# B&R Automation Studio project PT_KB_V01 (part 7)

#### TEHNICKI_DODATAK.md
~~~~markdown
# FLOW CHART MASTER — Rad_PG_KB + BRB2_rad

> Detaljni operativni dijagrami za state mašinu Podstanice Grejanja Kotlarnica Banja (PG_KB)
> i BRB2 (bunar) sa vezama preko AsIMA. Svi substepovi, tranzicije, akcije, timeouti.

---

## A. ASCII P&ID skica (referenca za sve dijagrame)

> **VAŽNO — topologija PG_PV05:** proporcionalni ventil `PG_PV05` je **odvojak PRE** `PG_V02` (ne posle). Odvaja se od dolazne BRB2 magistrale i vodi na drenažni kanal. `PG_V05` je zaseban ON/OFF ventil na bypass grani IEBKB1 — nema nikakve veze sa `PG_PV05`.

```
                    ┌── PG_PV05 ──> DRENAŽNI KANAL
                    │      • ispiranje: čeka T na TT_PG_07 >= 60 °C (SP podesiv sa HMI)
                    │      • održavanje pritiska ≥ 5 bar na potisu BRB2 dok su
                    │        ventili tanka zatvoreni (drži bunar u režimu)
                    │      • održavanje 6–7 bar dok su ventili tanka aktivni
                    │        (rasterećenje ka drenaži — štiti izmenjivače i cev)
                    │      • anti-hidraulički udar: P_dolaz > 6.5 bar → auto open
                    │
BRB2 ulaz ──────────┤
(optika ka BRB2_1)  │
                    │                          ┌─ PG_V06 ─ PG_PV01 ─┐
                    └── PG_V02 ────────────────┤                    ├──> Prihvatni tank
                                               └─ PG_V07 ─ PG_PV02 ─┘         │
                                                                              │  ┌ LS_PG_01 (nivo, SP=1.5m)
                                                                              │  ┌ PTNS_PG_01 (P,T,N)
                                                                              │
IEBKB1 ulaz ──> PG_V01 ──────────────> PG_V05 ────────────────────────────────┤
(optika ka IEBKB1)                    (BYPASS ON/OFF —                        │
                                       aktivan samo u IEBKB1 modu)            │
                                                                              │
                                                                       ┌── PG_V03 ── Pu_PG_01 ──┐
                                                                       │                        ├──> ka potrošačima
                                                                       └── PG_V04 ── Pu_PG_02 ──┘  (SP_PritisakPotisa)
```

**Senzori (logička imena u dokumentu → putanja u kodu):**

| Logičko ime | Putanja u kodu | Namena |
|---|---|---|
| `TT_PG_07` | `PG.Sens.Tt._4` (**NOVI — treba dodati u `PG_Sens_Tt_type`**) | Temperatura na drenažnoj cevi iza `PG_PV05` — uslov za završetak ispiranja (SP = 60 °C, podesiv sa HMI) |
| `PG_PT_dolaz` | `PG.Sens.Pt._1` | Pritisak termalne vode na ulazu u podstanicu (pre `PG_V02`) — uslov za anti-udar |
| `PG_PT_potis` | `PG.Sens.Pt._5` | Pritisak potisa iza pumpi `Pu_PG_01/02` (SP = `SetPritisakPotisa`) |
| `PG_PT_BRB2_potis` | `PG.Sens.Pt._6` | Dodatni transmiter -1..9 bar — pritisak dolazne magistrale iza `PG_V02` (mirror preko IMA ka BRB2) |
| `PG_FT_potis` | `PG.Sens.MP._1` | Protok potisa (za `MinProtok/MaxProtok` granice u varijanti 1) |
| `LS_PG_01` | `PG.Sens.LS._1` | Nizak nivo vode u prihvatnom tanku (SP = 1.5 m ciljno) |
| `PTNS_PG_01` | `PG.Sens.Pt._NS1` + `_NS2` | Pritisak na dnu (`_NS1`) i vrhu (`_NS2`) prihvatnog tanka (za proračun nivoa i P u vazdušnom prostoru) |

**Enumerisani selektori (RETAIN, definisani u [Types.typ](Types.typ)):**

| Selektor | Vrednosti |
|---|---|
| `SelektovaniIzvor` (`E_SelektovaniIzvor`) | `_00_nijedan`, `_01_BRB2`, `_02_IEBKB1` |
| `RegulacionaVarijanta` (`E_RegulacionaVarijanta`) | `_00_neaktivan`, `_01_REG_PRITISAK`, `_02_REG_PROTOK`, `_03_REG_TEMPERATURA` |
| `AktivnaPumpaIzlazTanka` (`E_AktivnaPumpaIzlazTanka`) | `_00_nijedna`, `_01_Pu_PG_01`, `_02_Pu_PG_02` |
| `AktivniPropVentilUlazTanka` (`E_AktivniPropVentilUlazTanka`) | `_00_nijedan`, `_01_PG_PV01`, `_02_PG_PV02` |

---

## B. PG_KB state mašina — detaljni stateDiagram

```mermaid
stateDiagram-v2
    direction TB

    [*] --> PG_00_Stand_By: cold boot (State default)

    state PG_00_Stand_By {
        [*] --> ST00_1
        ST00_1: 00.1 Verifikuj mirovanje sistema
        note right of ST00_1
            svi ventili CLOSED
            sve pumpe STOP
            SpremanZaBrb2 := FALSE
            SpremanZaIebkb1 := FALSE
        end note
    }

    PG_00_Stand_By --> PG_01_Priprema_BRB2: SelektovaniIzvor = _01_BRB2\nAND RegulacionaVarijanta <> _00_neaktivan\nAND KomandaStart
    PG_00_Stand_By --> PG_11_Priprema_IEBKB1: SelektovaniIzvor = _02_IEBKB1\nAND RegulacionaVarijanta <> _00_neaktivan\nAND KomandaStart

    %% ═══════════ GRANA BRB2 ═══════════
    state PG_01_Priprema_BRB2 {
        direction TB
        [*] --> ST01_1

        ST01_1: 01.1 Verifikacija interlockova
        note right of ST01_1
            check: PG_V01 = CLOSED
            check: PG_V06 = CLOSED, PG_V07 = CLOSED
            check: PG_V05 = CLOSED
            check: Pu_PG_01 = STOP, Pu_PG_02 = STOP
            check: PG_V03 = CLOSED, PG_V04 = CLOSED
            timeout 5s → Fault F01_INTERLOCK
        end note

        ST01_1 --> ST01_2: interlockovi OK

        ST01_2: 01.2 Otvaranje BRB2 dolaza + start ispiranja
        note right of ST01_2
            PG_V02 → OPEN
            PG_PV05 → 50% (drenaža otvorena)
            IMA: signal BRB2 = "start bunara u ispiranje modu (FR=20Hz)"
            čekaj potvrdu BRB2.PumpaAktivna = TRUE
            timeout 30s → Fault F02_BRB2_NEODZIVA
        end note

        ST01_2 --> ST01_3: BRB2 pumpa startovala

        ST01_3: 01.3 Čekanje temperature ispiranja
        note right of ST01_3
            monitor: TT_PG_07 >= SetPointMinTempIspiranja (60°C, podesivo sa HMI)
            trajanje ispiranja: obično 2-5 min
            timeout 10 min → Fault F03_ISPIRANJE_TIMEOUT
        end note

        ST01_3 --> ST01_4: T_dren dostigla SP

        ST01_4: 01.4 Preusmerenje na tank
        note right of ST01_4
            AKO AktivniPropVentilUlazTanka = _01_PG_PV01:
                PG_V06 → OPEN
                PG_PV01 → aktivan (regulacija nivoa tanka)
            AKO _02_PG_PV02:
                PG_V07 → OPEN
                PG_PV02 → aktivan
            pauza 2s (stabilizacija)
            PG_PV05 → 0% (zatvori drenažu)
            AKO AktivnaPumpaIzlazTanka = _01_Pu_PG_01:
                PG_V03 → OPEN
                Pu_PG_01 → START sa niskim FR (ramp up)
            AKO _02_Pu_PG_02:
                PG_V04 → OPEN
                Pu_PG_02 → START
        end note

        ST01_4 --> ST01_5: ventili otvoreni, pumpa startovala

        ST01_5: 01.5 Signal spremnosti
        note right of ST01_5
            čekaj: nivo tanka > 1.0 m (75% SP)
            čekaj: pritisak potisa >= 90% SP_PritisakPotisa
            čekaj: nema fault-ova
            SpremanZaBrb2 := TRUE
            IMA: šalji spremnost BRB2
        end note
    }

    PG_01_Priprema_BRB2 --> PG_02_Rad_BRB2: 01.5 OK → prelaz na rad
    PG_01_Priprema_BRB2 --> PG_03_Zaustavljanje_BRB2: Fault ILI KomandaStop

    state PG_02_Rad_BRB2 {
        direction TB
        [*] --> ST02_MAIN

        ST02_MAIN: 02.0 Regularni rad
        note right of ST02_MAIN
            aktivni PG_PV01/PV02 → PID(SetPointNivoTanka=1.5m)
            aktivna Pu_PG_01/02 → PID(SetPritisakPotisa)
            monitor MinProtok/MaxProtok override
            IMA: dvosmerni mirror stanja PG↔BRB2
        end note

        ST02_MAIN --> ST02_ANTI: P_dolaz > SetPointMaxPritisakDolaznaCev (6.5 bar)
        ST02_MAIN --> ST02_ROT: uslov rotacije pumpi (radni sati / manuelni zahtev)

        ST02_ANTI: 02.A Anti-hidraulički udar
        note right of ST02_ANTI
            PG_PV05 → auto otvaranje na drenažu (proporcionalno)
            trajanje: dok P_dolaz > 6.4 bar (histerezis 0.1)
            akcija u pozadini, ne menja stanje
        end note
        ST02_ANTI --> ST02_MAIN: P_dolaz < 6.4 bar (histerezis)

        ST02_ROT: 02.R Rotacija Pu_PG_01 ↔ Pu_PG_02
        note right of ST02_ROT
            OVERLAP tranzicija:
              1. start pratite pumpu na 0 Hz
              2. ramp up nova pumpa
              3. ramp down aktivna pumpa
              4. AktivnaPumpaIzlazTanka := novo
              5. zatvori stari PG_V03/V04
        end note
        ST02_ROT --> ST02_MAIN: rotacija završena
    }

    PG_02_Rad_BRB2 --> PG_03_Zaustavljanje_BRB2: KomandaStop\nILI Fault\nILI SelektovaniIzvor promena

    state PG_03_Zaustavljanje_BRB2 {
        direction TB
        [*] --> ST03_1

        ST03_1: 03.1 Redukcija protoka
        note right of ST03_1
            IMA: signal BRB2 = "ramp down bunara"
            PG_PV01/PV02 → ramp down otvor (5s)
            čekaj: protok < 10% MaxProtok
        end note

        ST03_1 --> ST03_2: protok nizak

        ST03_2: 03.2 Zatvaranje tank grane
        note right of ST03_2
            PG_V06 → CLOSED (ili PG_V07)
            PG_PV01 → 0% (ili PG_PV02)
            pauza 1s
        end note

        ST03_2 --> ST03_3: tank grana zatvorena

        ST03_3: 03.3 Zaustavljanje izlazne pumpe
        note right of ST03_3
            Pu_PG_01 → ramp down (ili Pu_PG_02)
            čekaj: pumpa STOP
            PG_V03 → CLOSED (ili PG_V04)
        end note

        ST03_3 --> ST03_4: izlaz zatvoren

        ST03_4: 03.4 Uslovno zatvaranje BRB2 dolaza
        note right of ST03_4
            AKO SelektovaniIzvor menja se u _02_IEBKB1:
                PG_V02 → CLOSED
                IMA: BRB2 = "stop bunara"
            AKO se izvor ne menja:
                PG_V02 ostaje OPEN (za brz restart)
                IMA: BRB2 = "stop bunara"
        end note
    }

    PG_03_Zaustavljanje_BRB2 --> PG_00_Stand_By: 03.4 OK, izvor se ne menja
    PG_03_Zaustavljanje_BRB2 --> PG_11_Priprema_IEBKB1: 03.4 OK, izvor promenjen u _02_IEBKB1

    %% ═══════════ GRANA IEBKB1 ═══════════
    state PG_11_Priprema_IEBKB1 {
        direction TB
        [*] --> ST11_1

        ST11_1: 11.1 Verifikacija interlockova
        note right of ST11_1
            check: PG_V02 = CLOSED
            check: PG_V06 = CLOSED, PG_V07 = CLOSED
            check: PG_PV05 = 0%
            check: PG_V05 = CLOSED
            check: PG_V03 = CLOSED, PG_V04 = CLOSED
            timeout 5s → Fault F11_INTERLOCK
        end note

        ST11_1 --> ST11_2: interlockovi OK

        ST11_2: 11.2 Otvaranje IEBKB1 grane
        note right of ST11_2
            PG_V01 → OPEN
            pauza 1s
            PG_V05 → OPEN (bypass ka tanku)
            IMA: signal IEBKB1 = "start pumpa sa zadatim protokom"
            čekaj potvrdu IEBKB1.PumpaAktivna
            timeout 30s → Fault F12_IEBKB1_NEODZIVA
        end note

        ST11_2 --> ST11_3: IEBKB1 pumpa startovala

        ST11_3: 11.3 Punjenje tanka
        note right of ST11_3
            monitor: nivo tanka raste
            čekaj: nivo >= 1.0 m (75% SP)
            timeout 5 min → Fault F13_PUNJENJE_TIMEOUT
        end note

        ST11_3 --> ST11_4: nivo dostignut

        ST11_4: 11.4 Start izlaza
        note right of ST11_4
            PG_V03 → OPEN (ili PG_V04)
            Pu_PG_01 → START (ili Pu_PG_02)
            čekaj: pritisak potisa >= 90% SP
            SpremanZaIebkb1 := TRUE
        end note
    }

    PG_11_Priprema_IEBKB1 --> PG_12_Rad_IEBKB1: 11.4 OK
    PG_11_Priprema_IEBKB1 --> PG_13_Zaustavljanje_IEBKB1: Fault ILI KomandaStop

    state PG_12_Rad_IEBKB1 {
        direction TB
        [*] --> ST12_MAIN

        ST12_MAIN: 12.0 Regularni rad IEBKB1
        note right of ST12_MAIN
            IEBKB1 pumpa gura zadati protok
            nivo tanka reguliše se protokom IEBKB1 (bez PG_PV01/PV02)
            PG_V05 stalno OPEN
            Pu_PG_01/02 → PID(SetPritisakPotisa)
            IMA: dvosmerni mirror stanja PG↔IEBKB1
        end note

        ST12_MAIN --> ST12_ROT: uslov rotacije izlaznih pumpi
        ST12_ROT: 12.R Rotacija Pu_PG_01 ↔ Pu_PG_02 (isti OVERLAP)
        ST12_ROT --> ST12_MAIN: rotacija završena
    }

    PG_12_Rad_IEBKB1 --> PG_13_Zaustavljanje_IEBKB1: KomandaStop\nILI Fault\nILI SelektovaniIzvor promena

    state PG_13_Zaustavljanje_IEBKB1 {
        direction TB
        [*] --> ST13_1

        ST13_1: 13.1 Redukcija protoka IEBKB1
        note right of ST13_1
            IMA: signal IEBKB1 = "ramp down pumpe"
            čekaj: protok < 10% MaxProtok
        end note

        ST13_1 --> ST13_2: protok nizak

        ST13_2: 13.2 Zatvaranje bypass
        note right of ST13_2
            PG_V05 → CLOSED
            pauza 1s
        end note

        ST13_2 --> ST13_3: bypass zatvoren

        ST13_3: 13.3 Zaustavljanje izlazne pumpe
        note right of ST13_3
            Pu_PG_01/02 → ramp down + STOP
            PG_V03/V04 → CLOSED
        end note

        ST13_3 --> ST13_4: izlaz zatvoren

        ST13_4: 13.4 Uslovno zatvaranje IEBKB1 dolaza
        note right of ST13_4
            AKO SelektovaniIzvor menja se u _01_BRB2:
                PG_V01 → CLOSED
            AKO se izvor ne menja:
                PG_V01 ostaje OPEN (za brz restart)
            IMA: IEBKB1 = "stop pumpa"
        end note
    }

    PG_13_Zaustavljanje_IEBKB1 --> PG_00_Stand_By: 13.4 OK, izvor se ne menja
    PG_13_Zaustavljanje_IEBKB1 --> PG_01_Priprema_BRB2: 13.4 OK, izvor promenjen u _01_BRB2

    %% ═══════════ AUTO-RESTART ═══════════
    note left of PG_00_Stand_By
        AUTO-RESTART posle nestanka struje:
        - State := PG_00_Stand_By (uvek)
        - Ako RETAIN.SelektovaniIzvor <> _00_nijedan
          I RETAIN.RegulacionaVarijanta <> _00_neaktivan
          → automatski KomandaStart → prelaz na 01/11
        - NE zatvara ventile koji su bili otvoreni pre restart-a
          (Priprema faza to prepoznaje kroz interlock check)
    end note
```

---

## C. BRB2_rad state mašina (podsetnik) — proširena Hotel + IEBKB1 grana

```mermaid
stateDiagram-v2
    direction TB

    [*] --> B00_StandBy: cold boot

    B00_StandBy --> B10_Priprema: KomandaStart (od PG_KB preko IMA)\nILI Priprema_Ispiranje

    state B10_Priprema {
        [*] --> B10_1
        B10_1: 10.1 Verifikacija RB2 interlockova
        B10_1 --> B10_2: OK
        B10_2: 10.2 Otvori RB2_V01 (dolaz sa bunara)
        B10_2 --> B10_3: OK
        B10_3: 10.3 Ispiranje (RB2 strana) - dok T_bunar OK
        B10_3 --> B10_4: T OK
        B10_4: 10.4 Grananje prema Ctrl.OdredisteBRB2
    }

    B10_Priprema --> B20_Rad_Hotel: OdredisteBRB2 = _01_Hotel
    B10_Priprema --> B25_Rad_IEBKB1: OdredisteBRB2 = _02_IEBKB1

    state B20_Rad_Hotel {
        [*] --> B20_1
        B20_1: 20.1 Otvori RB2_V02 (ka Hotelu preko PG)
        B20_1 --> B20_2: OK
        B20_2: 20.2 Ramp up pumpe bunara
        B20_2 --> B20_MAIN: OK
        B20_MAIN: 20.M Regularni rad prema RegulacionaVarijanta
        note right of B20_MAIN
            var _01_PRITISAK: FR = f(P_potis)
            var _02_PROTOK:  FR = f(FT_potis)
            var _03_TEMP:    FR = f(T_sekundar)
            IMA: dvosmerni mirror sa PG_KB
        end note
    }

    state B25_Rad_IEBKB1 {
        [*] --> B25_1
        B25_1: 25.1 Otvori RB2_V03 (ka IEBKB1)
        B25_1 --> B25_2: OK
        B25_2: 25.2 Ramp up pumpe bunara
        B25_2 --> B25_MAIN: OK
        B25_MAIN: 25.M Regularni rad za IEBKB1
        note right of B25_MAIN
            uvek varijanta protok
            FR = f(FT_potis)
        end note
    }

    B20_Rad_Hotel --> B30_Zaustavljanje_Hotel: KomandaStop ILI Fault
    B25_Rad_IEBKB1 --> B35_Zaustavljanje_IEBKB1: KomandaStop ILI Fault

    state B30_Zaustavljanje_Hotel {
        [*] --> B30_1
        B30_1: 30.1 Ramp down pumpa bunara
        B30_1 --> B30_2: FR = 0
        B30_2: 30.2 Zatvori RB2_V02
        B30_2 --> B30_3: OK
        B30_3: 30.3 Kondiciono zatvori RB2_V01
    }

    state B35_Zaustavljanje_IEBKB1 {
        [*] --> B35_1
        B35_1: 35.1 Ramp down pumpa
        B35_1 --> B35_2: FR = 0
        B35_2: 35.2 Zatvori RB2_V03
        B35_2 --> B35_3: OK
        B35_3: 35.3 Kondiciono zatvori RB2_V01
    }

    B30_Zaustavljanje_Hotel --> B00_StandBy
    B35_Zaustavljanje_IEBKB1 --> B00_StandBy

    %% Rotacija BRB2 ↔ BRB1_rez radi u pozadini, ne menja glavno stanje
    note left of B20_Rad_Hotel
        Rotacija BRB2 ↔ BRB1_rez:
        OVERLAP tranzicija, prati radne sate
        Menja Ctrl.AktivnaPumpaBunar bez zaustavljanja
    end note
```

---

## D. IMA komunikacija PG↔BRB2 — swimlane sekvenca (Priprema BRB2)

```mermaid
sequenceDiagram
    participant HMI as HMI Operator
    participant PG as PG_KB (PT_KB_V01)
    participant IMA as AsIMA link (optika)
    participant BRB as BRB2_rad (BRB2_1)

    Note over PG,BRB: Auto-boot ili KomandaStart

    HMI->>PG: Set SelektovaniIzvor=_01_BRB2, RegulacionaVarijanta=_02_REG_PROTOK
    HMI->>PG: Set AktivnaPumpaIzlazTanka=_01_Pu_PG_01
    HMI->>PG: Set AktivniPropVentilUlazTanka=_01_PG_PV01
    HMI->>PG: KomandaStart = TRUE

    PG->>PG: PG_00 → PG_01 (Priprema_BRB2)
    PG->>PG: ST01.1 verifikuj interlockove
    PG->>PG: ST01.2 OPEN PG_V02, PG_PV05=50%
    PG->>IMA: TX: Ctrl.SelektovaniIzvor, Ctrl.RegulacionaVarijanta, KomandaStart_BRB2
    IMA->>BRB: RX: Ctrl update od PG_KB

    BRB->>BRB: B00 → B10 (Priprema BRB2)
    BRB->>BRB: OPEN RB2_V01, start pumpa bunara FR=20Hz
    BRB->>IMA: TX: Status.PumpaAktivna=TRUE, Sens.FR_Bunar=20
    IMA->>PG: RX: Status BRB2

    PG->>PG: ST01.3 čekaj TT_PG_07 >= SetPointMinTempIspiranja (SP)
    PG->>IMA: TX: Sens.TT_PG_07 (svaki ciklus)
    IMA->>BRB: RX: (za HMI vizualizaciju na BRB strani)

    Note over PG: TT_PG_07 dostigla SP
    PG->>PG: ST01.4 OPEN PG_V06, PG_PV01 aktivan
    PG->>PG: ST01.4 CLOSE PG_PV05, OPEN PG_V03, START Pu_PG_01
    PG->>PG: ST01.5 SpremanZaBrb2 := TRUE
    PG->>IMA: TX: Status.SpremanZaBrb2=TRUE
    IMA->>BRB: RX: PG spreman

    BRB->>BRB: B10 → B20 (Rad Hotel) - ramp up FR
    BRB->>IMA: TX: Status.SpremanZaPodstanicu=TRUE

    PG->>PG: PG_01 → PG_02 (Rad BRB2)

    Note over PG,BRB: Regularni rad — sve se šalje na obe strane
    loop svaki ciklus
        PG->>IMA: TX: Sens.NivoTanka, PT_potis, FT_potis, TT_PG_07, PT_dolaz, PT_BRB2_potis
        PG->>IMA: TX: Act.Pu_PG_01_FR, PG_PV01_otvor, PG_PV05_otvor
        IMA->>BRB: RX (za HMI)
        BRB->>IMA: TX: Sens.FR_Bunar, PritisakBunar, ProtokBunar, TempBunar
        BRB->>IMA: TX: Act.Pumpa_bunar_snaga
        IMA->>PG: RX (za HMI)
    end
```

---

## E. Fault dijagram + Recovery putanje

```mermaid
stateDiagram-v2
    direction LR

    state "Normal Operation" as NORMAL {
        [*] --> RAD
        RAD: PG_02 / PG_12 aktivno
    }

    NORMAL --> F_INTERLOCK: interlock check FAIL u Priprema fazi
    NORMAL --> F_IZVOR: BRB2/IEBKB1 nije odgovorio 30s (IMA timeout)
    NORMAL --> F_ISPIRANJE: TT_PG_07 nije dostigla SP u 10 min
    NORMAL --> F_NIVO_HIGH: LS_PG_01 > 2.5 m (prepun tank)
    NORMAL --> F_NIVO_LOW: LS_PG_01 < 0.3 m u toku rada
    NORMAL --> F_PRITISAK_HIGH: P_dolaz > 8 bar u toku rada (iznad anti-udara)
    NORMAL --> F_PUMPA: Pu_PG_01/02 alarm (FB_HV_2LS status)
    NORMAL --> F_KOM_IMA: AsIMA link down > 5s

    state "Fault Handling" as FAULT {
        [*] --> F_KLASIFIKUJ
        F_KLASIFIKUJ: Klasifikuj tip fault-a
        F_KLASIFIKUJ --> F_HITNO: F_PRITISAK_HIGH ILI F_NIVO_HIGH
        F_KLASIFIKUJ --> F_KONTROL: F_INTERLOCK ILI F_IZVOR ILI F_KOM_IMA
        F_KLASIFIKUJ --> F_SOFT: F_ISPIRANJE ILI F_NIVO_LOW ILI F_PUMPA

        F_HITNO: HITNO — bezbedno zaustavljanje
        note right of F_HITNO
            SVI ventili CLOSED odmah
            SVE pumpe STOP odmah
            PG_PV05 OPEN (rasterećenje)
            State := PG_00_Stand_By
            FaultLatched := TRUE
            čeka ResetAllowed
        end note

        F_KONTROL: KONTROLISANO zaustavljanje
        note right of F_KONTROL
            prelaz na PG_03 ili PG_13
            uobičajena sekvenca zaustavljanja
            FaultLatched := TRUE
        end note

        F_SOFT: SOFT recovery
        note right of F_SOFT
            pauza u trenutnom substepu
            timeout retry 3x
            posle 3 neuspeha → F_KONTROL
        end note
    }

    F_INTERLOCK --> FAULT
    F_IZVOR --> FAULT
    F_ISPIRANJE --> FAULT
    F_NIVO_HIGH --> FAULT
    F_NIVO_LOW --> FAULT
    F_PRITISAK_HIGH --> FAULT
    F_PUMPA --> FAULT
    F_KOM_IMA --> FAULT

    FAULT --> NORMAL: ResetAllowed + KomandaReset od HMI

    note left of FAULT
        Sve klase pišu u FaultCode/FaultText
        Sve klase šalju IMA notifikaciju
        HMI dobija zvučni alarm
    end note
```

### E.1 Registar fault kodova (`FaultCode : USINT`)

| Kod | Klasa | Okidač | Akcija oporavka |
|-----|-------|--------|-----------------|
| `F01_INTERLOCK` | KONTROL | Interlock check fail u `PG_01` (BRB2 grana) — neki ventil nije u CLOSED, pumpe rade | Zaustavljanje kroz `PG_03` sekvencu; čeka `KomandaReset` |
| `F02_BRB2_NEODZIVA` | KONTROL | BRB2 pumpa nije potvrdila `PumpaAktivna` u 30 s (IMA timeout u `ST01_2`) | Prelaz `PG_03_Zaustavljanje_BRB2`, IMA notifikacija |
| `F03_ISPIRANJE_TIMEOUT` | SOFT | `TT_PG_07` nije dostigla SP (60 °C) u 10 min | Retry 3× (produžava `T_ispiranje`); posle 3. → KONTROL |
| `F11_INTERLOCK` | KONTROL | Interlock check fail u `PG_11` (IEBKB1 grana) | Zaustavljanje kroz `PG_13`; čeka reset |
| `F12_IEBKB1_NEODZIVA` | KONTROL | IEBKB1 pumpa nije potvrdila aktivnost u 30 s | `PG_13_Zaustavljanje_IEBKB1`, IMA notifikacija |
| `F13_PUNJENJE_TIMEOUT` | SOFT | Nivo tanka nije dostigao 1.0 m u 5 min tokom IEBKB1 punjenja | Retry 3×; posle 3. → KONTROL |
| `F20_NIVO_HIGH` | HITNO | `LS_PG_01` mapiran nivo > 2.5 m (prepun tank) | Svi ventili CLOSED, sve pumpe STOP, `PG_PV05` OPEN, State := `PG_00`, `FaultLatched := TRUE` |
| `F21_NIVO_LOW` | SOFT | `LS_PG_01` < 0.3 m u toku aktivnog rada | Pauza substepa, retry 3×; posle 3. → KONTROL |
| `F30_PRITISAK_HIGH` | HITNO | `PG_PT_dolaz` > 8 bar (iznad anti-udar praga 6.5) | HITNO gašenje kao `F20` |
| `F31_ANTI_UDAR_TRAJE` | SOFT | Anti-udar rasterećenje traje > 60 s bez pada P_dolaz-a | Retry 3×; posle 3. → KONTROL |
| `F40_PUMPA_PG` | SOFT | Alarm `Pu_PG_01/02` (FB_HV_2LS status) — pumpa ne prati komandu | Pauza, retry pokretanja; posle 3. → KONTROL sa rotacijom pumpi ako moguće |
| `F50_KOM_IMA` | KONTROL | AsIMA link down > 5 s | `PG_03/PG_13` kontrolisano gašenje; `FaultLatched` dok se link ne uspostavi + operater ne resetuje |
| `F60_KOM_BRB2` | KONTROL | Prijavljen `BRB2.FaultLatched = TRUE` preko IMA | `PG_03_Zaustavljanje_BRB2` |
| `F70_SENZOR_LOST` | HITNO | `ConfigValid = FALSE` na kritičnom `FBAI01_DI01` (Pt._1/._5/._6, MP._1, Tt._4) | HITNO gašenje |

**Reset uslovi:** `KomandaReset` sa HMI + `ResetAllowed = TRUE` (svi FB-ovi imaju `ResetAllowed` izlaz posle BR_Lib update-a).

---

## F. Mapa `.st` fajlova (nomenklatura per substep)

Predlažem sledeću strukturu (spremno za korak 3):

```
PT_KB_V01/Logical/Rad_PG_KB/
├── Cyclic.st                       (CASE dispečer - samo poziva substepove)
├── Init.st                          (default vrednosti SP-ova na cold boot)
├── Exit.st
├── Types.typ                        ✅ ažurirano
├── Variables.var
├── IEC.prg
└── Substeps/
    ├── PG_00_Stand_By.st
    ├── PG_01_1_Interlockovi.st
    ├── PG_01_2_Otvaranje_Ispiranje.st
    ├── PG_01_3_Cekanje_Temperature.st
    ├── PG_01_4_Preusmerenje_Tank.st
    ├── PG_01_5_Signal_Spreman.st
    ├── PG_02_Rad_BRB2.st
    ├── PG_02_A_Anti_Udar.st
    ├── PG_02_R_Rotacija_Pumpi.st
    ├── PG_03_1_Redukcija_Protoka.st
    ├── PG_03_2_Zatvaranje_Tank.st
    ├── PG_03_3_Zaustavljanje_Pumpe.st
    ├── PG_03_4_Uslovno_Zatvaranje_V02.st
    ├── PG_11_1_Interlockovi.st
    ├── PG_11_2_Otvaranje_Bypass.st
    ├── PG_11_3_Punjenje_Tanka.st
    ├── PG_11_4_Start_Izlaza.st
    ├── PG_12_Rad_IEBKB1.st
    ├── PG_13_1_Redukcija_Protoka.st
    ├── PG_13_2_Zatvaranje_Bypass.st
    ├── PG_13_3_Zaustavljanje_Pumpe.st
    ├── PG_13_4_Uslovno_Zatvaranje_V01.st
    ├── FAULT_Klasifikator.st
    ├── FAULT_Hitno.st
    ├── FAULT_Kontrol.st
    └── FAULT_Soft.st
```

Cyclic.st tada postaje kratak dispatcher:

```pascal
CASE State OF
    PG_00_Stand_By:           PG_00_Stand_By_Body();
    PG_01_Priprema_BRB2:
        CASE Substep OF
            1: PG_01_1_Interlockovi();
            2: PG_01_2_Otvaranje_Ispiranje();
            3: PG_01_3_Cekanje_Temperature();
            4: PG_01_4_Preusmerenje_Tank();
            5: PG_01_5_Signal_Spreman();
        END_CASE;
    (* ... itd ... *)
END_CASE;

(* Fault se poziva iznad state mašine kao gate *)
IF FaultLatched THEN
    FAULT_Klasifikator();
END_IF;
```

---

## G. Sledeći koraci (nakon što potvrdiš dijagrame)

1. ~~**Korak 1**: definicija tipova i strukture upravljačkog konteksta.~~ **✅ URAĐENO**
    `E_RegulacionaVarijanta`, `E_SelektovaniIzvor`, `E_AktivnaPumpaIzlazTanka`, `E_AktivniPropVentilUlazTanka`, `typParPG` i `typCtrlPG` su deo globalnog tipa `PG_type`; paralelno `typBRB2Rad` postoji u [BRB2_1/Logical/Project/BRB2_rad/Types.typ](../../../../BRB2_1/Logical/Project/BRB2_rad/Types.typ). `PG : PG_type` i `BRB2Rad : typBRB2Rad` deklarisani su kao `RETAIN`.
2. ~~**Korak 2**: preusmeriti postojeći `Cyclic.st` da koristi `PG.Ctrl.*` umesto pojedinačnih promenljivih.~~ **✅ URAĐENO** (i za `BRB2_rad/Cyclic.sfc`).
3. **Korak 2.5** (na redu): dopuna [Variables.var](Variables.var):
   - `Substep : USINT := 0` (0 = ulazak u state, 1..N = koraci)
   - `KomandaStart : BOOL`, `KomandaStop : BOOL`, `KomandaReset : BOOL` (sa HMI)
   - `FaultLatched : BOOL`
   - `FaultCode : USINT` (šifre iz sekcije E.1)
   - `FaultText : STRING[80]` (za HMI display)
   - Dodati `T_OverlapPumpi : TIME := T#10s` u `typParPG_KB` u [Types.typ](Types.typ)
4. **Korak 2.6** (paralelno): dodati u `PG_Sens_Tt_type` u [Global.typ](../Global.typ) novo polje `_4 : FBAI01_DI01;` sa komentarom „Temperatura na drenaznoj cevi iza PG_PV05 — TT_PG_07", plus fizičko mapiranje kanala u [IO](../IO/).
5. **Korak 3**: kreirati folder `Substeps/` sa praznim skeletonima svakog substep fajla (imena iz sekcije F).
6. **Korak 4**: kreirati komunikacioni tip `PG_00_Comm_Types.typ` — čisto-podatkovni mirror struct (samo `REAL`/`BOOL`/`INT`, bez FB instanci) za AsIMA prenos u oba smera. Poštuje BR_Lib verzijsku razliku između BRB2_1 i PT_KB_V01.
7. **Korak 5**: implementirati logiku redom (najsigurniji prvo — `PG_00_Stand_By`, pa `PG_01_1_Interlockovi`, itd.).
8. **Korak 6**: sinhronizovati enum ekvivalente i mirror strukture u BRB2_1 (za simetriju IMA).

---

## H. Zatvorena pitanja iz validacije dijagrama

| # | Pitanje | Odluka |
|---|---------|--------|
| 1 | Nazivi senzora (`PG_TT_dren`, `PG_PT_dolaz`…) | Prihvaćeno mapiranje iz sekcije A tabele senzora. Kanonska imena u kodu su `PG.Sens.Pt._N` / `Tt._N` / `MP._1` / `LS._N`; logička imena (`TT_PG_07`, `PG_PT_dolaz`, itd.) su za HMI i dokumentaciju. |
| 2 | Fault klase HITNO / KONTROL / SOFT | Prihvaćeno. Detaljan registar u sekciji E.1. |
| 3 | OVERLAP tranzicija pumpi — parametar? | **Da**, `T_OverlapPumpi : TIME := T#10s` dodaje se u `typParPG_KB` (Korak 2.5). Isto važi za rotaciju bunarskih pumpi u `typParBRB2Rad`. |
| 4 | Tip `Substep` varijable — `USINT` ili posebna enum? | `USINT` (0..255). Numeracija prati oznake u sekciji B (npr. `PG_01_1` → `Substep = 1`). Jednostavnije nego enum po fazi, i kompatibilno sa CASE dispečerom u [Cyclic.st](Cyclic.st). |

---

## I. Trenutno stanje implementacije (baseline)

**Legenda:** ✅ postoji u kodu · 🟡 delimično · ⛔ nedostaje

### I.1 PT_KB_V01 / `Rad_PG_KB`

| Artifakt | Fajl | Status |
|---|---|---|
| `E_PG_KB_State` | [Types.typ](Types.typ) | ✅ |
| `E_RegulacionaVarijanta` | [Types.typ](Types.typ) | ✅ |
| `E_SelektovaniIzvor` | [Types.typ](Types.typ) | ✅ |
| `E_AktivnaPumpaIzlazTanka` | [Types.typ](Types.typ) | ✅ |
| `E_AktivniPropVentilUlazTanka` | [Types.typ](Types.typ) | ✅ |
| `typParPG_KB` (Par) | [Types.typ](Types.typ) | ✅ (nedostaje `T_OverlapPumpi`) |
| `typCtrlPG_KB` (Ctrl) | [Types.typ](Types.typ) | ✅ |
| `typPG_KB` | [Types.typ](Types.typ) | ✅ |
| `PG_KB : typPG_KB` (RETAIN) | [Variables.var](Variables.var) | ✅ |
| `State : E_PG_KB_State` | [Variables.var](Variables.var) | ✅ |
| `Substep : USINT` | [Variables.var](Variables.var) | ⛔ Korak 2.5 |
| `KomandaStart/Stop/Reset : BOOL` | [Variables.var](Variables.var) | ⛔ Korak 2.5 |
| `FaultLatched, FaultCode, FaultText` | [Variables.var](Variables.var) | ⛔ Korak 2.5 |
| `Cyclic.st` koristi `PG.Ctrl.*` | [Cyclic.st](Cyclic.st) | ✅ (samo grananje `SelektovaniIzvor`; nema substep dispečera) |
| Substep dispečer (CASE po substep-u) | [Cyclic.st](Cyclic.st) | ⛔ Korak 3 |
| Substep fajlovi u `Substeps/` | — | ⛔ Korak 3 |

### I.2 PT_KB_V01 / globalni tipovi

| Artifakt | Fajl | Status |
|---|---|---|
| `PG_Sens_Pt_type._1.._6, _NS1/2` | [Global.typ](../Global.typ) | ✅ |
| `PG_Sens_Tt_type._1.._3` | [Global.typ](../Global.typ) | ✅ |
| `PG_Sens_Tt_type._4` (TT_PG_07) | [Global.typ](../Global.typ) | ⛔ Korak 2.6 |
| `PG_Sens_MP_type._1` | [Global.typ](../Global.typ) | ✅ |
| `PG_Sens_LS_type._1.._5` | [Global.typ](../Global.typ) | ✅ |

### I.3 BRB2_1 / `BRB2_rad`

| Artifakt | Fajl | Status |
|---|---|---|
| `E_RegulacionaVarijanta` | `BRB2_1/Logical/Project/BRB2_rad/Types.typ` | ✅ |
| `typParBRB2Rad` / `typCtrlBRB2Rad` / `typBRB2Rad` | `BRB2_1/Logical/Project/BRB2_rad/Types.typ` | ✅ |
| `BRB2Rad : typBRB2Rad` (RETAIN) | `BRB2_1/Logical/Project/BRB2_rad/Variables.var` | ✅ |
| `Cyclic.sfc` koristi `BRB2Rad.Ctrl.OdredisteBRB2` | `BRB2_1/Logical/Project/BRB2_rad/Cyclic.sfc` | ✅ |
| `T_OverlapPumpi` (rotacija bunarskih pumpi) | `typParBRB2Rad` | ⛔ Korak 2.5 |
| SFC koraci sa stvarnom logikom | `BRB2_1/Logical/Project/BRB2_rad/Cyclic.sfc` | 🟡 (koraci definisani, sadržaj prazan) |
| BR_Lib verzija (`FB_HV_2LS`, `FB_DI`, `FB_V_ON_OFF_FB`) | `BRB2_1/Logical/Libraries/BR_Lib` | 🟡 stara — treba upgrade pre AsIMA mirror-a (vidi Korak 4) |

### I.4 AsIMA komunikacija PG ↔ BRB2

| Artifakt | Status |
|---|---|
| Fizička optička veza (hardware) | ✅ |
| AsIMA konfiguracija u AS projektu | ⛔ Korak 4 |
| `PG_00_Comm_Types.typ` (mirror struct) | ⛔ Korak 4 |
| Slanje/prijem po ciklusu iz Cyclic-a | ⛔ Korak 4 |

---
~~~~

#### FLOW_CHART_PITANJA.md
```markdown
# Pitanja za flow chart obe strane (BRB2 + PT_KB_V01)

> Upiši odgovore direktno ispod svakog pitanja (na liniji `Odgovor:`).
> Ono što još nisi odlučio ostavi prazno — o tome ćemo posle razgovarati.
> Kad završiš, samo javi "spremno".

---

## FAZA 3: PT_KB_V01 STRANA, GRANA BRB2

### 3.1 `PG_01_Priprema_BRB2`

Šta se sve mora desiti pre nego što Podstanica "objavi" da je spremna za BRB2 (dozvola BRB2 startu)?

**a) Koji ventili se otvaraju/zatvaraju u pripremi?**
(npr. PG_V01 dolazni od BRB2, PG_V02 ka tanku, PG_V03/PG_V04 na izlazu iz tanka — koji od ovih se dira ovde?)

Odgovor: pojsanio u drugom fajlu

**b) Koja pumpa izlaza iz tanka (Pu_PG_01 ili Pu_PG_02) se startuje u pripremi ili tek u fazi Rad_BRB2?**

Odgovor: sve pojasnjeno kada je tank u rau pupa se pali kad nivo predje preko 1.5 metara a gasi kada nivo padne ispod 0.9 metara - ako odrzava nivo ako odzava pritisak ne interesuje je nivo dok ne padne ispod miniumam onda krece da odrzava taj minimalni nivo

**c) Ima li provera pritiska/temperature pre nego što se izađe iz Priprema?**

Odgovor:odgovrio u drugom fajlu

**d) Koji "OK" signal Podstanica šalje BRB2 strani preko IMA (npr. `PG.Status.SpremanZaBrb2 : BOOL`) — i šta znači?**

Odgovor:odgovreno ranije

---

### 3.2 `PG_02_Rad_BRB2`

Šta radi Podstanica dok BRB2 aktivno gura vodu?

**a) Koja pumpa izlaza iz tanka radi (Pu_PG_01 default? auto rotacija? manual?)**

Odgovor:odogovreno vec

**b) Za trenutno aktivnu Varijantu 2 (BRB2 vodi, PG samo prazni tank do nivoa):**
Koji je "nivo" za regulaciju? Nivo tanka (LT_ senzor)? Pritisak potisa PG pumpe? Nešto treće?

Odgovor:odgovoreno

**c) Šta se dešava sa Varijantom 1 (PG vodi, prati pritisak):**
Ako je aktivna, da li PG šalje "traži više/manje" komandu BRB2 strani preko IMA?

Odgovor:odgovoreno - salje samo nivo i status

**d) Da li se PG_V03/PG_V04 preključuju u toku rada (rotacija pumpe za istrošivost)?**

Odgovor: verovatnio resavacemo kasnije

---

### 3.3 `PG_03_Zaustavljanje_BRB2`

Šta radi Podstanica kada operater (ili sistem) povuče izvor (`SelektovaniIzvor = _00_`)?

**a) Da li Podstanica prvo zaustavlja svoju izlaznu pumpu, pa BRB2 pumpu? Ili obratno? Ili paralelno?**

Odgovor:odgovoreno

**b) Ventili koji se zatvaraju u ovoj fazi — redosled?**

Odgovor: odgovreno ranije

**c) Kada je Zaustavljanje "završeno" — koji su uslovi za povratak u Stand_By?**
(svi ventili zatvoreni? pumpe stopped? pritisak spao ispod X bar?)

Odgovor:odgovreno ranije

---

## FAZA 3.5: PRELAZ Pu_PG_01 ↔ Pu_PG_02

**3.5.a Kako se odlučuje koja pumpa je aktivna?**
Označi ono što važi (obriši ostalo, ili kombinuj):
- [ ] manual (operater sa HMI)
- [ ] auto rotacija po vremenu rada
- [ ] auto rotacija po broju startovanja
- [ ] fallback na drugu ako prva ima alarm
- [ ] kombinacija (dopiši kakva)

Odgovor:odgovreno ranije

**3.5.b Prelaz mora imati "overlap" (obe pumpe rade kratko) ili "hard switch" (jedna se ugasi pre nego druga krene)?**

Odgovor:odgovreno ranije

**3.5.c Ventili PG_V03/PG_V04 — da li se ikad obe drže zatvorene (npr. dok pumpe stoje) ili je barem jedan uvek otvoren?**

Odgovor:odgovreno ranije

---

## FAZA 2: BRB2 STRANA, IEBKB1 GRANA (B25 / B35 / B45)

**2.a Da li je logika ista kao Hotel grana (isti ramp, isti pritisci) samo drugi ventili (RB1_V01 vs RB1_V02, RB2_V01 vs RB2_V02)?**

Odgovor:odgovreno ranije

**2.b Ako je različita — šta se razlikuje?**
(npr. drugi `P_Target`, drugi flush režim, drugi `FR_RampUp`)

Odgovor:nista

**2.c Ispiranje (`IspiranjeAktivno` + PG_PV05) — da li se izvodi za obe grane isto ili samo za Hotel?**

Odgovor:odgovreno ranije

---

## FAZA 4: PT_KB_V01 STRANA, GRANA IEBKB1

**4.a Postoji li već legacy kod (u nekom projektu koji nam nije trenutno otvoren) koji rukuje IEBKB1 stranom sa PT_KB_V01 tačke?**

Odgovor:odgovreno ranije

**4.b Ako ne, samo skiciraj u par rečenica šta se treba desiti (u kojoj se meri razlikuje od BRB2 grane).**

Odgovor:odgovreno ranije

---

## FAULT / PREKIDNE PUTANJE

**F.a Ako se javi kritični fault (npr. LT tanka izgubljen, flow meter izgubljen) u toku `Rad_BRB2` — da li:**
- [ ] sistem preskače direktno u `Zaustavljanje_BRB2` sa normalnom sekvencom
- [ ] postoji zaseban Fault step (`PG_99_Fault`) sa agresivnim gašenjem
- [ ] operater mora ručno da povuče izvor pa da krene normalno gašenje

Odgovor:odgovreno ranije

**F.b Ista pitanja za BRB2 stranu (fault tokom `B30_RadBrb2Hotel`):**

Odgovor:odgovreno ranije

---

## BONUS PITANJE ZA MAPIRANJE

**M.a Da li već imaš fizički nacrtan PID/PFD dijagram procesa (PDF/DWG/scan) koji ti mogu pogledati radi validacije naziva ventila i tokova?**
Ako da, gde ga mogu naći?

Odgovor:odgovreno ranije
```

#### FLOW_CHART_POJASNJENJA.md
~~~~markdown
# Pojašnjenja pre finalnih flow chart-ova

> 6 kratkih pitanja koja su izronila iz tvojih odgovora.
> Popuni pored svakog, snimi, i javi „spremno".

---

## P1. PG_V06 / PG_V07 — potvrda semantike

Iz odgovora zaključujem:
- **PG_V06** = ON/OFF ventil PRE proporcionalnog **PG_PV01**
- **PG_V07** = ON/OFF ventil PRE proporcionalnog **PG_PV02**

Da li je to tačno? Ako nije, kako se zovu i za šta služe?

Odgovor: da tacno je

---

## P2. PG_PV05 — dvostruka uloga?

Do sada je `PG_PV05` bio pomenut kao proporcionalni ventil za **ispiranje/drenažu** (na BRB2 strani, `IspiranjeAktivno`).

Ali sada u odgovoru za pripremu BRB2 kažeš: „pušta se bunar dok voda **na drenaži iza PG_PV05** ne dođe do ~60°C".

Da li je to isti PG_PV05, ili postoji poseban drenažni put? Da li se u pripremi otvara `PG_PV05` na drenažu prema kojem procenatu?

Odgovor:da to je isti venti i on radi isto sto i ventili na ulaz u tank odrzava poritisak na potisu iz BRB2 preko 5 bara uvek ... osim kad su aktivni vetili na ulazu u tank tada on odrzava pritisak na 6 ilio 7 bara i cuva iouzmenjivace i celu liniju od velikog pritiska

---

## P3. Signal PG → BRB2 preko IMA

Šta sve konkretno PG šalje BRB2 strani preko IMA (i obratno)?

Trenutno pretpostavljam PG → BRB2:
- `SpremanZaBrb2 : BOOL`
- `NivoTanka : REAL`
- `RegulacionaVarijanta : E_RegulacionaVarijanta`
- `SelektovaniIzvor : E_SelektovaniIzvor` (ogledalo)

BRB2 → PG:
- `Pt_6_Pressure : REAL` (pritisak dolazne cevi, čita se lokalno u BRB2)
- `Pu_Aktivna : BOOL` (BRB2 pumpa aktivna)
- `FR_Actual : REAL` (trenutna frekvencija BRB2 pumpe)
dodaj i protok ka hotelu
mada je meni ovde biola ideja da se salje sve na obe strane takod a mozes da pridjes izuelizaciji i da ividis i jednu i drugu stranu ....
jer ima protokol je mocan a mi imamo optiku nista necemo ugroziti a dacemo lepu komciju u radu na terenu

Fali/suvišno/preimenovati?

Odgovor: dat gore

---

## P4. Aktivna pumpa BRB2

Rekao si: "postoji logika u kodu kako pumpa radi kada je sistem aktivan, pogledaj, jednostavno je i imaš već i parametre unutra — javi šta si našao".

Našao sam ove parametre u `BRB2_1/Logical/Project/BRB2_rad/Types.typ`:

```
FR_Start        : REAL := 20.0;  (* startna frekvenca [Hz] *)
FR_RampUp       : REAL := 0.5;   (* ramp up [Hz/s] *)
FR_RampDown     : REAL := 0.25;  (* ramp down [Hz/s] *)
T_Zaletanje     : TIME := T#10s; (* pre pocetka podizanja *)
P_Target        : REAL := 5.0;   (* ciljni pritisak Pt_RB2_2 [bar] *)
P_TargetStop    : REAL := 5.2;   (* stop pritisak [bar] *)
FR_MinZeroFlow  : REAL := 0.0;   (* TODO eksperimentalno *)
MinProtok       : REAL;          (* Var1 donja granica *)
MaxProtok       : REAL;          (* Var1 gornja granica *)
SetProtok       : REAL := 6.0;   (* Var2 zadati protok [l/s] *)
```

**Ali gore si u odgovoru 3.1.b rekao "samo treba da se pali selektovana pumpa, sad radi logika samo na pumpu koja je povezana"** — ovo se odnosi na **BRB2 pumpu** (jedna pumpa) ili na **PG izlaz pumpu** (Pu_PG_01/Pu_PG_02)?

Odgovor: odnosi se na PG 01/02

---

## P5. Auto-restart posle nestanka struje

Ovo je važno za dizajn. Predlog:

Kada se PLC probudi:
- `State := PG_00_Stand_By` (uvek?)
- Ili: pročitaj RETAIN `SelektovaniIzvor` i idi u odgovarajući step ako je bio aktivan?

Ako je bio aktivan (npr. `SelektovaniIzvor = _01_BRB2` pre nestanka struje), da li:

- [ ] auto-vrati sistem u `PG_02_Rad_BRB2` bez ponovne pripreme (rizik: ventili u nepoznatom stanju)
- [ ] prođi kroz `PG_01_Priprema_BRB2` sa svim proverama pa u `PG_02_Rad_BRB2`
- [ ] uđi u posebno **Recovery** stanje koje polako obnavlja proces sa proverama pritisaka

Odgovor: vracas se us tanje stand By i pokreces sistem sa preselektovanim ocijama
ne zatvaras PG_PV02 jer se nemanja izvor npr ...

---

## P6. PID dijagram — ponovo pošalji

Rekao si da si mi već poslao PID dijagram. Ako je bio u prethodnoj sesiji, nemam ga trenutno pri ruci.

Molim te:
1. Ubaci ga u chat **kao attachment (slika)** — direktno ću ga pročitati i validirati imena ventila
2. ILI ga stavi u fajl u projektu i reci mi putanju

Odgovor / putanja:

---dodao u prilog

## Šta ću uraditi paralelno (bez čekanja)

Dok odgovaraš, ja radim ovo:

1. **Dodajem `E_AktivniPropVentilUlazTanka` u `typCtrlPG_KB`** (analogno `AktivnaPumpaIzlazTanka`).
2. **Dodajem `SetPointNivoTanka : REAL := 1.5` u `typParPG_KB`**.
3. Pravim **`FLOW_CHART_MASTER.md`** sa mermaid dijagramima:
   - Nadgradnja PG_KB state masine (isti tvoj E_PG_KB_State ali sada sa svim substepima)
   - Isto za BRB2_rad (E_BRB2_State — proširenje trenutnog SFC-a u ST logiku)
   - Sekvenca komunikacije PG↔BRB2 preko IMA
   - Fault putanja + Recovery putanja

Kada odgovoriš na P1–P6, dopunjujem sve rupe i dobijamo finalni dokument koji je „ground truth" za dalju implementaciju.
~~~~

#### FLOW_CHART_POJASNJENJA_2.md
~~~~markdown
# Poslednje mikro-nejasnoće pre finalnog dijagrama

> Popuni pored svakog, snimi, javi "spremno" — pa krećem sa flow chartom.

---

## ISPRAVLJENO RAZUMEVANJE (posle korisnikovih korekcija)

- **PG_PV05** = proporcionalni ventil DIREKTNO na drenažnoj grani (nema ON/OFF ventila pre njega). Uloge:
  - početno **ispiranje** cevi (dok voda ne postigne 60°C na drenaži)
  - **zaštita od hidrauličkih udara** / rasterećenje visokog pritiska (prag ~6.5 bar)
- **PG_V05** = ON/OFF ventil na potpuno posebnoj **bypass grani** za IEBKB1 mod (zaobilazi PG_PV01/PV02, pušta direktno u tank). NEMA VEZE sa PG_PV05.

Topologija:
```
                          ┌── PG_PV05 ──> DRENAŽA
BRB2 ulaz ──> PG_V02 ─────┼── PG_V06 ──> PG_PV01 ──> tank
                          └── PG_V07 ──> PG_PV02 ──> tank
                                                       ▲
IEBKB1 ulaz ──> PG_V01 ────────────> PG_V05 ───────────┘  (bypass)
```pg PV05 se odvaja pre dolaka BRB2 do PG_V02 pogledaj PID !!! ipravi to

---

## PZ1. Anti-udar prag za PG_PV05

Rekao si "6.5 bar". Interpretiram kao: kada pritisak u dolaznoj magistrali (posle PG_V02) pređe 6.5 bar, PG_PV05 se automatski otvara na drenažu radi rasterećenja.

Odgovor: 6.5 Bara

---

## PZ2. PG_V05 — ON/OFF ventil (iz IEBKB1 odgovora)

U odgovoru za IEBKB1 granu si rekao: "otvaraš PG_V01 i PG_V05".

Na PID-u vidim `PG_V05` blizu tanka. Da li je to:
- ON/OFF ventil iza PG_PV05 (posle proporcionalnog, pre ulaska u tank drugim putem)?
- ON/OFF ventil na bypass liniji koja u IEBKB1 modu zaobilazi PG_PV01/PV02?
- Nešto treće?

Kada se otvara PG_V05? U kom modu (samo IEBKB1? i BRB2 nekad?)

Odgovor: - ON/OFF ventil na bypass liniji koja u IEBKB1 modu zaobilazi PG_PV01/PV02?

---

## PZ3. Temperatura drenaže (60°C uslov)

Kada prelaziš sa IEBKB1 na BRB2, BRB2 bunar startuje i "izbacuje" hladnu vodu kroz drenažu dok ne postigne 60°C.

Pitanja:
- Gde je senzor temperature? Koje je ime PG_TT_XX?
- Kroz koji put ide drenaža — kroz PG_PV05 pa gde?
- Koji ventil se otvara na drenažu za vreme grejanja? (Da li je to `PG_V22` sa tanka? Ili nešto drugo?)
- Da li BRB2 pumpa radi u konstantnoj frekvenci tokom ove faze (npr. 20-30 Hz) ili prati neki cilj?

Odgovor: treba das e ugradi objasnio ranije gde se ugradjuje - nbegde na drenaznu cev gde moze da meri temperaturu bode u drenaznoj cevi
Kroz PV05 pa and renzani kanal ucrtano u PID-u i ta temperatura trba da bude SP koji se moze menjati
~~~~

### Program Logical/PG_Intf (IEC)

#### Cyclic.st
```iecst
PROGRAM _CYCLIC
	(* ======================================================================== *)
	(* 1) Lokalni PT-BRB2 procesni ugovor                                       *)
	(* ======================================================================== *)
	PGRad_BRB2.RadKaPodstanici := PGRad_BRB2Cmd.RadKaPodstanici;
	PGRad_BRB2.ManualMode := PGRad_BRB2Cmd.ManualMode;
	PGRad_BRB2.ManualSequence := PGRad_BRB2Cmd.ManualSequence;
	PGRad_BRB2.ManualStart := PGRad_BRB2Cmd.ManualStart;
	PGRad_BRB2.ManualStop := PGRad_BRB2Cmd.ManualStop;
	PGRad_BRB2.ManualNextStep := PGRad_BRB2Cmd.ManualNextStep;
	PGRad_BRB2.ManualAbort := PGRad_BRB2Cmd.ManualAbort;
	PGRad_BRB2.ZahtevStarta := PGRad_BRB2Cmd.ZahtevStarta;
	PGRad_BRB2.ZahtevZaustavljanja := PGRad_BRB2Cmd.ZahtevZaustavljanja;
	PGRad_BRB2.VentiliPodstaniceZatvoreni := PGRad_BRB2Cmd.VentiliPodstaniceZatvoreni;
	PGRad_BRB2.PritisakIEBKB1 := PGRad_BRB2Cmd.PritisakIEBKB1;
	PGRad_BRB2.PodstanicaURezimuRada := PGRad_BRB2Cmd.PodstanicaURezimuRada;

	(* ======================================================================== *)
	(* 2) PT izlazni AsIMA snapshot                                             *)
	(* ======================================================================== *)
	PGRad_BRB2_Tx.RadKaPodstanici := PGRad_BRB2Cmd.RadKaPodstanici;
	PGRad_BRB2_Tx.ManualMode := PGRad_BRB2Cmd.ManualMode;
	PGRad_BRB2_Tx.ManualSequence := PGRad_BRB2Cmd.ManualSequence;
	PGRad_BRB2_Tx.ManualStart := PGRad_BRB2Cmd.ManualStart;
	PGRad_BRB2_Tx.ManualStop := PGRad_BRB2Cmd.ManualStop;
	PGRad_BRB2_Tx.ManualNextStep := PGRad_BRB2Cmd.ManualNextStep;
	PGRad_BRB2_Tx.ManualAbort := PGRad_BRB2Cmd.ManualAbort;
	PGRad_BRB2_Tx.ZahtevStarta := PGRad_BRB2Cmd.ZahtevStarta;
	PGRad_BRB2_Tx.ZahtevZaustavljanja := PGRad_BRB2Cmd.ZahtevZaustavljanja;
	PGRad_BRB2_Tx.VentiliPodstaniceZatvoreni := PGRad_BRB2Cmd.VentiliPodstaniceZatvoreni;
	PGRad_BRB2_Tx.PritisakIEBKB1 := PGRad_BRB2Cmd.PritisakIEBKB1;
	PGRad_BRB2_Tx.PodstanicaURezimuRada := PGRad_BRB2Cmd.PodstanicaURezimuRada;

	(* ======================================================================== *)
	(* 3) BRB2 ulazni procesni status                                           *)
	(* ======================================================================== *)
	PGRad_BRB2.PumpaAktivna := PGRad_BRB2_Rx.PumpaAktivna;
	PGRad_BRB2.IspiranjeProtokDostignut := PGRad_BRB2_Rx.IspiranjeProtokDostignut;
	PGRad_BRB2.IspiranjeMinTrajanjeDostignuto := PGRad_BRB2_Rx.IspiranjeMinTrajanjeDostignuto;
	PGRad_BRB2.StopSPDostignut := PGRad_BRB2_Rx.StopSPDostignut;
	PGRad_BRB2.RB2V01Zatvoren := PGRad_BRB2_Rx.RB2V01Zatvoren;
	PGRad_BRB2.RB2V02Zatvoren := PGRad_BRB2_Rx.RB2V02Zatvoren;
END_PROGRAM
```

#### Exit.st
```iecst
PROGRAM _EXIT
END_PROGRAM
```

#### Init.st
```iecst
PROGRAM _INIT
END_PROGRAM
```

### Program Logical/HMI_Svc (IEC)

#### Init.st - Init code
```iecst
PROGRAM _INIT
	(* ======================================================================== *)
	(* 1) Inicijalizacija Podstanica trend prikaza                              *)
	(* ======================================================================== *)
	PGRad_TrendCursor.Position := 0.5;
	PGRad_TrendCursor.ViewSpan := 14400;
	PGRad_TrendCursor.PreviousViewSpan := 14400;
	PGRad_TrendCursor.FollowNow := TRUE;
	PGRad_TrendCursor.CmdBack := FALSE;
	PGRad_TrendCursor.CmdForward := FALSE;
	PGRad_TrendCursor.CmdNow := FALSE;
END_PROGRAM
```

#### Cyclic.st - Cyclic code
```iecst
PROGRAM _CYCLIC
	(* ======================================================================== *)
	(* 1) Rezim i raspolozivi vremenski opseg Podstanica trenda                 *)
	(* ======================================================================== *)
	(* VC pri otvaranju continuous trenda postavlja mod 1; mod 0 drzi zadati prozor. *)
	PGRad_TrendCursor.AxisMode := 0;

	TrendClock.enable := TRUE;
	TrendClock();
	TrendNow_s := DT_TO_UDINT(TrendClock.DT1);
	IF TrendNow_s > 864000 THEN
		TrendEarliest_s := TrendNow_s - 864000;
	ELSE
		TrendEarliest_s := 0;
	END_IF;
	IF (DT_TO_UDINT(PGRad_TrendCursor.RecordingStart) > TrendEarliest_s)
		AND (DT_TO_UDINT(PGRad_TrendCursor.RecordingStart) <= TrendNow_s) THEN
		TrendEarliest_s := DT_TO_UDINT(PGRad_TrendCursor.RecordingStart);
	END_IF;

	(* ======================================================================== *)
	(* 2) Zoom i navigacija vremenskog prozora                                  *)
	(* ======================================================================== *)
	IF PGRad_TrendCursor.ViewSpan < 3600 THEN
		PGRad_TrendCursor.ViewSpan := 3600;
	ELSIF PGRad_TrendCursor.ViewSpan > 172800 THEN
		PGRad_TrendCursor.ViewSpan := 172800;
	END_IF;

	IF (DT_TO_UDINT(PGRad_TrendCursor.ViewStart) = 0)
		AND (TrendNow_s >= DINT_TO_UDINT(PGRad_TrendCursor.ViewSpan)) THEN
		PGRad_TrendCursor.ViewStart := UDINT_TO_DT(
			TrendNow_s - DINT_TO_UDINT(PGRad_TrendCursor.ViewSpan));
		PGRad_TrendCursor.FollowNow := FALSE;
	END_IF;

	IF PGRad_TrendCursor.ViewSpan <> PGRad_TrendCursor.PreviousViewSpan THEN
		IF PGRad_TrendCursor.FollowNow THEN
			PGRad_TrendCursor.ViewStart := UDINT_TO_DT(
				TrendNow_s - DINT_TO_UDINT(PGRad_TrendCursor.ViewSpan));
		ELSE
			PGRad_TrendCursor.ViewStart := UDINT_TO_DT(
				DT_TO_UDINT(PGRad_TrendCursor.ViewStart)
				+ DINT_TO_UDINT(PGRad_TrendCursor.PreviousViewSpan)
				- DINT_TO_UDINT(PGRad_TrendCursor.ViewSpan));
		END_IF;
		PGRad_TrendCursor.PreviousViewSpan := PGRad_TrendCursor.ViewSpan;
		PGRad_TrendCursor.FollowNow := FALSE;
	END_IF;

	IF PGRad_TrendCursor.CmdNow THEN
		IF TrendNow_s >= DINT_TO_UDINT(PGRad_TrendCursor.ViewSpan) THEN
			PGRad_TrendCursor.ViewStart := UDINT_TO_DT(
				TrendNow_s - DINT_TO_UDINT(PGRad_TrendCursor.ViewSpan));
		END_IF;
		PGRad_TrendCursor.FollowNow := FALSE;
	END_IF;

	IF PGRad_TrendCursor.CmdBack THEN
		PGRad_TrendCursor.FollowNow := FALSE;
		IF DT_TO_UDINT(PGRad_TrendCursor.ViewStart) > (TrendEarliest_s + DINT_TO_UDINT(PGRad_TrendCursor.ViewSpan)) THEN
			PGRad_TrendCursor.ViewStart := UDINT_TO_DT(
				DT_TO_UDINT(PGRad_TrendCursor.ViewStart) - DINT_TO_UDINT(PGRad_TrendCursor.ViewSpan));
		ELSE
			PGRad_TrendCursor.ViewStart := UDINT_TO_DT(TrendEarliest_s);
		END_IF;
	END_IF;

	IF PGRad_TrendCursor.CmdForward THEN
		IF (DT_TO_UDINT(PGRad_TrendCursor.ViewStart) + (2 * DINT_TO_UDINT(PGRad_TrendCursor.ViewSpan))) >= TrendNow_s THEN
			PGRad_TrendCursor.ViewStart := UDINT_TO_DT(
				TrendNow_s - DINT_TO_UDINT(PGRad_TrendCursor.ViewSpan));
			PGRad_TrendCursor.FollowNow := FALSE;
		ELSE
			PGRad_TrendCursor.ViewStart := UDINT_TO_DT(
				DT_TO_UDINT(PGRad_TrendCursor.ViewStart) + DINT_TO_UDINT(PGRad_TrendCursor.ViewSpan));
		END_IF;
	END_IF;

	(* ======================================================================== *)
	(* 3) Oznake vremenske ose i apsolutno vreme kursora                        *)
	(* ======================================================================== *)
	PGRad_TrendCursor.AxisTime0 := PGRad_TrendCursor.ViewStart;
	PGRad_TrendCursor.AxisTime1 := UDINT_TO_DT(
		DT_TO_UDINT(PGRad_TrendCursor.ViewStart) + (DINT_TO_UDINT(PGRad_TrendCursor.ViewSpan) / 8));
	PGRad_TrendCursor.AxisTime2 := UDINT_TO_DT(
		DT_TO_UDINT(PGRad_TrendCursor.ViewStart) + ((2 * DINT_TO_UDINT(PGRad_TrendCursor.ViewSpan)) / 8));
	PGRad_TrendCursor.AxisTime3 := UDINT_TO_DT(
		DT_TO_UDINT(PGRad_TrendCursor.ViewStart) + ((3 * DINT_TO_UDINT(PGRad_TrendCursor.ViewSpan)) / 8));
	PGRad_TrendCursor.AxisTime4 := UDINT_TO_DT(
		DT_TO_UDINT(PGRad_TrendCursor.ViewStart) + ((4 * DINT_TO_UDINT(PGRad_TrendCursor.ViewSpan)) / 8));
	PGRad_TrendCursor.AxisTime5 := UDINT_TO_DT(
		DT_TO_UDINT(PGRad_TrendCursor.ViewStart) + ((5 * DINT_TO_UDINT(PGRad_TrendCursor.ViewSpan)) / 8));
	PGRad_TrendCursor.AxisTime6 := UDINT_TO_DT(
		DT_TO_UDINT(PGRad_TrendCursor.ViewStart) + ((6 * DINT_TO_UDINT(PGRad_TrendCursor.ViewSpan)) / 8));
	PGRad_TrendCursor.AxisTime7 := UDINT_TO_DT(
		DT_TO_UDINT(PGRad_TrendCursor.ViewStart) + ((7 * DINT_TO_UDINT(PGRad_TrendCursor.ViewSpan)) / 8));
	PGRad_TrendCursor.AxisTime8 := UDINT_TO_DT(
		DT_TO_UDINT(PGRad_TrendCursor.ViewStart) + DINT_TO_UDINT(PGRad_TrendCursor.ViewSpan));

	(* VC vraca vreme kursora u ms od pocetka referentnog trend zapisa. *)
	PGRad_TrendCursor.DateTime := UDINT_TO_DT(
		DT_TO_UDINT(PGRad_TrendCursor.RecordingStart)
		+ (PGRad_TrendCursor.Time / 1000));

	PGRad_TrendCursor.CmdBack := FALSE;
	PGRad_TrendCursor.CmdForward := FALSE;
	PGRad_TrendCursor.CmdNow := FALSE;
END_PROGRAM
```

### Package Logical/ProcessUnit - Funkcionalne procesne jedinice.

### Program Logical/ProcessUnit/ProcUnit (IEC)

#### Init.st - Init code
```iecst
PROGRAM _INIT
	(* AirRelease parametri se inicijalizuju u vlasnickom Rad_PG_KB sloju. *)
END_PROGRAM
```

#### Cyclic.st - Cyclic code
```iecst
PROGRAM _CYCLIC
	(* ======================================================================== *)
	(* PROCUNIT - ODZRACIVANJE BR1 I BR2                                     *)
	(* AUTO: FB_AirRelease vodi pritisak i LS stepene.                        *)
	(* MANUAL: EnableManual i ManualSP_Percent daju direktnu servisnu komandu. *)
	(* STOP/FAULT: reset, alarm i bezbedno zatvaranje ostaju u vlasnistvu FB-a. *)
	(* STATUS: State, Alarm, Position i Fault statusi se objavljuju HMI-ju.   *)
	(* ======================================================================== *)
	(* ======================================================================== *)
	(* 1) Izbor parametara odzracivanja prema aktivnom izvoru                   *)
	(* ======================================================================== *)
	IF PGRad_Cmd.AirRelease.UseIEBKB1Parameters THEN
		PGRad_AirRelease.PV03.FB.AR_Param := PGRad.Par.AirRelease.IEBKB1.PV03;
		PGRad_AirRelease.PV04.FB.AR_Param := PGRad.Par.AirRelease.IEBKB1.PV04;
	ELSE
		PGRad_AirRelease.PV03.FB.AR_Param := PGRad.Par.AirRelease.BRB2.PV03;
		PGRad_AirRelease.PV04.FB.AR_Param := PGRad.Par.AirRelease.BRB2.PV04;
	END_IF;

	(* ======================================================================== *)
	(* 2) PV03 odzracivanje ulaza u podstanicu                                  *)
	(* ======================================================================== *)
	PGRad_AirRelease.PV03.FB.AR_Input.Enable := PGRad_Cmd.AirRelease.PV03.Enable;
	PGRad_AirRelease.PV03.FB.AR_Input.EnableManual := PGRad_AirRelease.PV03.Ctrl.EnableManual;
	PGRad_AirRelease.PV03.FB.AR_Input.ManualSP_Percent := PGRad_AirRelease.PV03.Ctrl.ManualSP_Percent;
	PGRad_AirRelease.PV03.FB.AR_Input.Pressure_bar := PG.Sens.Pt._1.AI_Output.ScaledValue;
	PGRad_AirRelease.PV03.FB.AR_Input.LS1_Upper := PG.Sens.LS._3.DI_Output.Value;
	PGRad_AirRelease.PV03.FB.AR_Input.LS2_Middle := PG.Sens.LS._2.DI_Output.Value;
	PGRad_AirRelease.PV03.FB.AR_Input.LS3_Lower := FALSE;
	PGRad_AirRelease.PV03.FB.AR_Input.ResetAlarm :=
		PGRad_Cmd.AirRelease.ResetAll
		OR PGRad_AirRelease.PV03.Ctrl.ResetAlarm
		OR (PT_Alarm.ResetPulse.Devices AND PGRad_AirRelease.PV03.FB.AR_Output.ResetAllowed);
	PGRad_AirRelease.PV03.FB();
	PGRad_AirRelease.PV03.Ctrl.ResetAlarm := FALSE;

	(* ======================================================================== *)
	(* 3) PV04 odzracivanje ulaza u prihvatni tank                              *)
	(* ======================================================================== *)
	PGRad_AirRelease.PV04.FB.AR_Input.Enable := PGRad_Cmd.AirRelease.PV04.Enable;
	PGRad_AirRelease.PV04.FB.AR_Input.EnableManual := PGRad_AirRelease.PV04.Ctrl.EnableManual;
	PGRad_AirRelease.PV04.FB.AR_Input.ManualSP_Percent := PGRad_AirRelease.PV04.Ctrl.ManualSP_Percent;
	PGRad_AirRelease.PV04.FB.AR_Input.Pressure_bar := PG.Sens.Pt._4.AI_Output.ScaledValue;
	PGRad_AirRelease.PV04.FB.AR_Input.LS1_Upper := PG.Sens.LS._5.DI_Output.Value;
	PGRad_AirRelease.PV04.FB.AR_Input.LS2_Middle := PG.Sens.LS._4.DI_Output.Value;
	PGRad_AirRelease.PV04.FB.AR_Input.LS3_Lower := FALSE;
	PGRad_AirRelease.PV04.FB.AR_Input.ResetAlarm :=
		PGRad_Cmd.AirRelease.ResetAll
		OR PGRad_AirRelease.PV04.Ctrl.ResetAlarm
		OR (PT_Alarm.ResetPulse.Devices AND PGRad_AirRelease.PV04.FB.AR_Output.ResetAllowed);
	PGRad_AirRelease.PV04.FB();
	PGRad_AirRelease.PV04.Ctrl.ResetAlarm := FALSE;
END_PROGRAM
```

#### Exit.st - Exit code
```iecst
PROGRAM _EXIT
	(* ProcessUnit nema resurse koje treba zatvarati. *)
END_PROGRAM
```

### Package Logical/IMA_comm_PG_BRB2 - AsIMA master veza podstanice sa BRB2.

### Program Logical/IMA_comm_PG_BRB2/BRB2_com (IEC)

#### Init.st - Init code
```iecst
PROGRAM _INIT
	ResetCommunication := FALSE;
	ResetInProgress := FALSE;
	ResetDone := FALSE;
	ResetFault := FALSE;
	(* ======================================================================== *)
	(* 1) Otvaranje AsIMA master sesije prema BRB2                               *)
	(* ======================================================================== *)
	(* Ime DataObject-a identifikuje AsIMA server BRB2 i vraca stationId sesije. *)
	pDatObjName := ADR('BRB2');
	statusInit := IMAinit(pDatObjName, errorInfo, ADR(stationId));
END_PROGRAM
```

#### Cyclic.st - Cyclic code
```iecst
PROGRAM _CYCLIC
	(* ======================================================================== *)
	(* 1) Priprema i prenos PG01 lokalnog snapshot-a                            *)
	(* ======================================================================== *)
	(* PublishPG01 priprema lokalni AsIMA DTO; IMAcomm obavlja dvosmerni prenos. *)
	IF statusInit = IMA_OK THEN
		PublishPG01;
		statusComm := IMAcomm(stationId, connInfoPV, connInfoAUX);
	END_IF

	(* ======================================================================== *)
	(* 2) Automatsko brisanje komunikacione greske                              *)
	(* ======================================================================== *)
	(* ClearError se zadaje samo dok AsIMA prijavljuje gresku ili povezivanje. *)
	IF (connInfoPV.connectionStatus = IMA_ERROR)
		OR (connInfoPV.connectionStatus = IMA_CONNECTING) THEN
		connInfoPV.commandClearError := 1;
	ELSE
		connInfoPV.commandClearError := 0;
	END_IF

	PG01_Remote := PG01_Remote;
END_PROGRAM
```

#### Exit.st - Exit code
```iecst
PROGRAM _EXIT
	(* ======================================================================== *)
	(* 1) Zatvaranje otvorene AsIMA master sesije                                *)
	(* ======================================================================== *)
	(* Sesija se zatvara samo kada je INIT uspesno dodelio vazeci stationId. *)
	IF stationId <> 0 THEN
		statusClose := IMAclose(stationId);
	END_IF
END_PROGRAM
```

#### Variables.var - Local variables
```iecst
VAR
	(* AsIMA DataObject i identifikator sesije. *)
	pDatObjName : UDINT;       (* Adresa naziva AsIMA DataObject konfiguracije. *)
	stationId : UDINT;         (* Identifikator master AsIMA sesije. *)

	(* Povratni statusi AsIMA poziva. *)
	statusInit : UINT;         (* Rezultat jednokratne AsIMA inicijalizacije. *)
	statusComm : UINT;         (* Rezultat ciklicnog AsIMA prenosa. *)
	statusClose : UINT;        (* Rezultat zatvaranja AsIMA sesije. *)

	(* Dijagnostika inicijalizacije i PV prenosa. *)
	errorInfo : imaInfoStruct; (* Dijagnostika neuspele inicijalizacije. *)
	connInfoPV : imaInfoStruct; (* Status i dijagnostika PV prenosa ka BRB2. *)
	connInfoAUX : imaInfoStruct; (* Status pomocnih AsIMA servisa. *)
	ResetCommunication : BOOL; (* HMI zahtev za ponovno otvaranje AsIMA sesije. *)
	ResetInProgress : BOOL; (* Ponovna inicijalizacija AsIMA sesije je u toku. *)
	ResetDone : BOOL; (* Poslednja HMI reinicijalizacija je uspesno zavrsena. *)
	ResetFault : BOOL; (* Poslednja HMI reinicijalizacija nije uspela. *)
END_VAR
```

#### PublishPG01.st
```iecst
ACTION PublishPG01:
	(* ======================================================================== *)
	(* PUBLISH_PG01 - STATUSNI SNAPSHOT PODSTANICE ZA ASIMA/HMI               *)
	(* AUTO/MANUAL: samo objavljuje izabrane komande i statuse; ne komanduje   *)
	(* lokalnim aktuatorima. STOP/FAULT se prenose kao statusi i kodovi.       *)
	(* ======================================================================== *)
	(* ======================================================================== *)
	(* 1) PG01 kontrolni snapshot za AsIMA DTO                                  *)
	(* ======================================================================== *)
	(* Lokalna stanja se pretvaraju u stabilne brojcane vrednosti komunikacionog ugovora. *)
	(* 1.1) Izabrani izvor termalne vode. *)
	CASE PGRad.Ctrl.SelektovaniIzvor OF
		_01_BRB2: PG01_Local.PGCtrl.Izvor := 1;
		_02_IEBKB1: PG01_Local.PGCtrl.Izvor := 2;
	ELSE
		PG01_Local.PGCtrl.Izvor := 0;
	END_CASE

	(* 1.2) Izabrana regulaciona varijanta izlazne pumpe. *)
	CASE PGRad.Ctrl.RegulacionaVarijanta OF
		_01_REG_PRITISAK: PG01_Local.PGCtrl.Regulacija := 1;
		_02_REG_NIVO: PG01_Local.PGCtrl.Regulacija := 2;
	ELSE
		PG01_Local.PGCtrl.Regulacija := 0;
	END_CASE

	(* 1.3) Izabrana izlazna pumpa prihvatnog tanka. *)
	CASE PGRad.Ctrl.AktivnaPumpaIzlazTanka OF
		_01_Pu_PG_01: PG01_Local.PGCtrl.IzlaznaPumpa := 1;
		_02_Pu_PG_02: PG01_Local.PGCtrl.IzlaznaPumpa := 2;
	ELSE
		PG01_Local.PGCtrl.IzlaznaPumpa := 0;
	END_CASE

	(* 1.4) Aktivni proporcionalni ventil na ulazu tanka. *)
	CASE PGRad.Ctrl.AktivniPropVentilUlazTanka OF
		_01_PG_PV01: PG01_Local.PGCtrl.UlazniPV := 1;
		_02_PG_PV02: PG01_Local.PGCtrl.UlazniPV := 2;
	ELSE
		PG01_Local.PGCtrl.UlazniPV := 0;
	END_CASE

	PG01_Local.PGCtrl.AutoRestart := PGRad.Ctrl.AutoRestart;
	PG01_Local.PGCtrl.State := PGRad_Status.State;
	PG01_Local.PGCtrl.Substep := PGRad_Status.Substep;
	PG01_Local.PGCtrl.Fault := PGRad_Status.Fault;
	PG01_Local.PGCtrl.FaultCode := PGRad_Status.FaultCode;

	(* ======================================================================== *)
	(* 2) PG01 lokalni snapshot za AsIMA sinoptiku                              *)
	(* ======================================================================== *)
	(* 2.1) Pu01: komanda, ostvareni rad, frekvencija i fault prve izlazne pumpe. *)
	PG01_Local.PGAct.Pu01.RunCmd := PG.Act.Pu._1.Start;
	PG01_Local.PGAct.Pu01.Running := PG.Act.Pu._1.Status_inRun;
	PG01_Local.PGAct.Pu01.Frequency := PG.Act.Pu._1.Ostvarena_brzina;
	PG01_Local.PGAct.Pu01.Alarm := PG.Act.Pu._1.Alarm_FR OR PG.Act.Pu._1.Alarm_CAN;

	(* 2.2) Pu02: komanda, ostvareni rad, frekvencija i fault druge izlazne pumpe. *)
	PG01_Local.PGAct.Pu02.RunCmd := PG.Act.Pu._2.Start;
	PG01_Local.PGAct.Pu02.Running := PG.Act.Pu._2.Status_inRun;
	PG01_Local.PGAct.Pu02.Frequency := PG.Act.Pu._2.Ostvarena_brzina;
	PG01_Local.PGAct.Pu02.Alarm := PG.Act.Pu._2.Alarm_FR OR PG.Act.Pu._2.Alarm_CAN;

	(* 2.3) PV01 i PV02: komandovana i stvarna pozicija ulaznih ventila tanka. *)
	PG01_Local.PGAct.PV01.Enable := PG.Act.PV._1.PV_Input.Enable;
	PG01_Local.PGAct.PV01.CmdPercent := PG.Act.PV._1.PV_Output.ActiveSP_Percent;
	PG01_Local.PGAct.PV01.PositionPercent := PG.Act.PV._1.PV_Output.PV_Percent;
	PG01_Local.PGAct.PV01.Alarm := PG.Act.PV._1.PV_Output.FaultActive;
	PG01_Local.PGAct.PV02.Enable := PG.Act.PV._2.PV_Input.Enable;
	PG01_Local.PGAct.PV02.CmdPercent := PG.Act.PV._2.PV_Output.ActiveSP_Percent;
	PG01_Local.PGAct.PV02.PositionPercent := PG.Act.PV._2.PV_Output.PV_Percent;
	PG01_Local.PGAct.PV02.Alarm := PG.Act.PV._2.PV_Output.FaultActive;
	(* 2.4) PV03, PV04 i PV05: lokalni status ostalih proporcionalnih ventila. *)
	PG01_Local.PGAct.PV03.Enable := PG.Act.PV._3.PV_Input.Enable;
	PG01_Local.PGAct.PV03.CmdPercent := PG.Act.PV._3.PV_Output.ActiveSP_Percent;
	PG01_Local.PGAct.PV03.PositionPercent := PG.Act.PV._3.PV_Output.PV_Percent;
	PG01_Local.PGAct.PV03.Alarm := PG.Act.PV._3.PV_Output.FaultActive;
	PG01_Local.PGAct.PV04.Enable := PG.Act.PV._4.PV_Input.Enable;
	PG01_Local.PGAct.PV04.CmdPercent := PG.Act.PV._4.PV_Output.ActiveSP_Percent;
	PG01_Local.PGAct.PV04.PositionPercent := PG.Act.PV._4.PV_Output.PV_Percent;
	PG01_Local.PGAct.PV04.Alarm := PG.Act.PV._4.PV_Output.FaultActive;
	PG01_Local.PGAct.PV05.Enable := PG.Act.PV._5.PV_Input.Enable;
	PG01_Local.PGAct.PV05.CmdPercent := PG.Act.PV._5.PV_Output.ActiveSP_Percent;
	PG01_Local.PGAct.PV05.PositionPercent := PG.Act.PV._5.PV_Output.PV_Percent;
	PG01_Local.PGAct.PV05.Alarm := PG.Act.PV._5.PV_Output.FaultActive;

	(* 2.5) AV01 i AV02: dvosmerne komande i granicni prekidaci dovodnih ventila. *)
	PG01_Local.PGAct.AV01.OpenCmd := PG.Act.AV._1.V_Output.CmdOpen;
	PG01_Local.PGAct.AV01.CloseCmd := PG.Act.AV._1.V_Output.CmdClose;
	PG01_Local.PGAct.AV01.Opened := PG.Act.AV._1.Opened;
	PG01_Local.PGAct.AV01.Closed := PG.Act.AV._1.Closed;
	PG01_Local.PGAct.AV01.Alarm := PG.Act.AV._1.V_Output.FaultLatched;
	PG01_Local.PGAct.AV02.OpenCmd := PG.Act.AV._2.V_Output.CmdOpen;
	PG01_Local.PGAct.AV02.CloseCmd := PG.Act.AV._2.V_Output.CmdClose;
	PG01_Local.PGAct.AV02.Opened := PG.Act.AV._2.Opened;
	PG01_Local.PGAct.AV02.Closed := PG.Act.AV._2.Closed;
	PG01_Local.PGAct.AV02.Alarm := PG.Act.AV._2.V_Output.FaultLatched;
	(* 2.6) AV03 do AV07: zahtev otvaranja, polozaj i fault procesnih ventila. *)
	PG01_Local.PGAct.AV03.OpenCmd := PG.Act.AV._3.Open;
	PG01_Local.PGAct.AV03.Opened := PG.Act.AV._3.Opened;
	PG01_Local.PGAct.AV03.Closed := PG.Act.AV._3.Closed;
	PG01_Local.PGAct.AV03.Alarm := PG.Act.AV._3.V_Output.FaultLatched;
	PG01_Local.PGAct.AV04.OpenCmd := PG.Act.AV._4.Open;
	PG01_Local.PGAct.AV04.Opened := PG.Act.AV._4.Opened;
	PG01_Local.PGAct.AV04.Closed := PG.Act.AV._4.Closed;
	PG01_Local.PGAct.AV04.Alarm := PG.Act.AV._4.V_Output.FaultLatched;
	PG01_Local.PGAct.AV05.OpenCmd := PG.Act.AV._5.Open;
	PG01_Local.PGAct.AV05.Opened := PG.Act.AV._5.Opened;
	PG01_Local.PGAct.AV05.Closed := PG.Act.AV._5.Closed;
	PG01_Local.PGAct.AV05.Alarm := PG.Act.AV._5.V_Output.FaultLatched;
	PG01_Local.PGAct.AV06.OpenCmd := PG.Act.AV._6.Open;
	PG01_Local.PGAct.AV06.Opened := PG.Act.AV._6.Opened;
	PG01_Local.PGAct.AV06.Closed := PG.Act.AV._6.Closed;
	PG01_Local.PGAct.AV06.Alarm := PG.Act.AV._6.V_Output.FaultLatched;
	PG01_Local.PGAct.AV07.OpenCmd := PG.Act.AV._7.Open;
	PG01_Local.PGAct.AV07.Opened := PG.Act.AV._7.Opened;
	PG01_Local.PGAct.AV07.Closed := PG.Act.AV._7.Closed;
	PG01_Local.PGAct.AV07.Alarm := PG.Act.AV._7.V_Output.FaultLatched;
	(* 2.7) RV19 i RV21 do RV27: samo fizicki polozaj i alarm rucnih ventila. *)
	PG01_Local.PGAct.RV19.Opened := PG.Act.RV._19.HV_Output.Opened;
	PG01_Local.PGAct.RV19.Closed := PG.Act.RV._19.HV_Output.Closed;
	PG01_Local.PGAct.RV19.Alarm := PG.Act.RV._19.HV_Output.AlarmLatched;
	PG01_Local.PGAct.RV21.Opened := PG.Act.RV._21.HV_Output.Opened;
	PG01_Local.PGAct.RV21.Closed := PG.Act.RV._21.HV_Output.Closed;
	PG01_Local.PGAct.RV21.Alarm := PG.Act.RV._21.HV_Output.AlarmLatched;
	PG01_Local.PGAct.RV22.Opened := PG.Act.RV._22.HV_Output.Opened;
	PG01_Local.PGAct.RV22.Closed := PG.Act.RV._22.HV_Output.Closed;
	PG01_Local.PGAct.RV22.Alarm := PG.Act.RV._22.HV_Output.AlarmLatched;
	PG01_Local.PGAct.RV23.Opened := PG.Act.RV._23.HV_Output.Opened;
	PG01_Local.PGAct.RV23.Closed := PG.Act.RV._23.HV_Output.Closed;
	PG01_Local.PGAct.RV23.Alarm := PG.Act.RV._23.HV_Output.AlarmLatched;
	PG01_Local.PGAct.RV24.Opened := PG.Act.RV._24.HV_Output.Opened;
	PG01_Local.PGAct.RV24.Closed := PG.Act.RV._24.HV_Output.Closed;
	PG01_Local.PGAct.RV24.Alarm := PG.Act.RV._24.HV_Output.AlarmLatched;
	PG01_Local.PGAct.RV25.Opened := PG.Act.RV._25.HV_Output.Opened;
	PG01_Local.PGAct.RV25.Closed := PG.Act.RV._25.HV_Output.Closed;
	PG01_Local.PGAct.RV25.Alarm := PG.Act.RV._25.HV_Output.AlarmLatched;
	PG01_Local.PGAct.RV26.Opened := PG.Act.RV._26.HV_Output.Opened;
	PG01_Local.PGAct.RV26.Closed := PG.Act.RV._26.HV_Output.Closed;
	PG01_Local.PGAct.RV26.Alarm := PG.Act.RV._26.HV_Output.AlarmLatched;
	PG01_Local.PGAct.RV27.Opened := PG.Act.RV._27.HV_Output.Opened;
	PG01_Local.PGAct.RV27.Closed := PG.Act.RV._27.HV_Output.Closed;
	PG01_Local.PGAct.RV27.Alarm := PG.Act.RV._27.HV_Output.AlarmLatched;

	(* 2.8) Pritisci: vrednost, validnost i fault za svaki analogni Pt kanal. *)
	PG01_Local.PGSens.Pt00.Value := PG.Sens.Pt._0_0.AI_Output.ScaledValue;
	PG01_Local.PGSens.Pt00.Valid := PG.Sens.Pt._0_0.AI_Output.Status;
	PG01_Local.PGSens.Pt00.Alarm := PG.Sens.Pt._0_0.AI_Output.FaultLatched;
	PG01_Local.PGSens.Pt01.Value := PG.Sens.Pt._1.AI_Output.ScaledValue;
	PG01_Local.PGSens.Pt01.Valid := PG.Sens.Pt._1.AI_Output.Status;
	PG01_Local.PGSens.Pt01.Alarm := PG.Sens.Pt._1.AI_Output.FaultLatched;
	PG01_Local.PGSens.Pt02.Value := PG.Sens.Pt._2.AI_Output.ScaledValue;
	PG01_Local.PGSens.Pt02.Valid := PG.Sens.Pt._2.AI_Output.Status;
	PG01_Local.PGSens.Pt02.Alarm := PG.Sens.Pt._2.AI_Output.FaultLatched;
	PG01_Local.PGSens.Pt03.Value := PG.Sens.Pt._3.AI_Output.ScaledValue;
	PG01_Local.PGSens.Pt03.Valid := PG.Sens.Pt._3.AI_Output.Status;
	PG01_Local.PGSens.Pt03.Alarm := PG.Sens.Pt._3.AI_Output.FaultLatched;
	PG01_Local.PGSens.Pt04.Value := PG.Sens.Pt._4.AI_Output.ScaledValue;
	PG01_Local.PGSens.Pt04.Valid := PG.Sens.Pt._4.AI_Output.Status;
	PG01_Local.PGSens.Pt04.Alarm := PG.Sens.Pt._4.AI_Output.FaultLatched;
	PG01_Local.PGSens.Pt05.Value := PG.Sens.Pt._5.AI_Output.ScaledValue;
	PG01_Local.PGSens.Pt05.Valid := PG.Sens.Pt._5.AI_Output.Status;
	PG01_Local.PGSens.Pt05.Alarm := PG.Sens.Pt._5.AI_Output.FaultLatched;
	PG01_Local.PGSens.Pt06.Value := PG.Sens.Pt._6.AI_Output.ScaledValue;
	PG01_Local.PGSens.Pt06.Valid := PG.Sens.Pt._6.AI_Output.Status;
	PG01_Local.PGSens.Pt06.Alarm := PG.Sens.Pt._6.AI_Output.FaultLatched;
	PG01_Local.PGSens.PtNS1.Value := PG.Sens.Pt._NS1.AI_Output.ScaledValue;
	PG01_Local.PGSens.PtNS1.Valid := PG.Sens.Pt._NS1.AI_Output.Status;
	PG01_Local.PGSens.PtNS1.Alarm := PG.Sens.Pt._NS1.AI_Output.FaultLatched;
	PG01_Local.PGSens.PtNS2.Value := PG.Sens.Pt._NS2.AI_Output.ScaledValue;
	PG01_Local.PGSens.PtNS2.Valid := PG.Sens.Pt._NS2.AI_Output.Status;
	PG01_Local.PGSens.PtNS2.Alarm := PG.Sens.Pt._NS2.AI_Output.FaultLatched;
	(* 2.9) Temperature: vrednost, validnost i fault za svaki analogni Tt kanal. *)
	PG01_Local.PGSens.Tt01.Value := PG.Sens.Tt._1.AI_Output.ScaledValue;
	PG01_Local.PGSens.Tt01.Valid := PG.Sens.Tt._1.AI_Output.Status;
	PG01_Local.PGSens.Tt01.Alarm := PG.Sens.Tt._1.AI_Output.FaultLatched;
	PG01_Local.PGSens.Tt02.Value := PG.Sens.Tt._2.AI_Output.ScaledValue;
	PG01_Local.PGSens.Tt02.Valid := PG.Sens.Tt._2.AI_Output.Status;
	PG01_Local.PGSens.Tt02.Alarm := PG.Sens.Tt._2.AI_Output.FaultLatched;
	PG01_Local.PGSens.Tt03.Value := PG.Sens.Tt._3.AI_Output.ScaledValue;
	PG01_Local.PGSens.Tt03.Valid := PG.Sens.Tt._3.AI_Output.Status;
	PG01_Local.PGSens.Tt03.Alarm := PG.Sens.Tt._3.AI_Output.FaultLatched;
	PG01_Local.PGSens.Tt04.Value := PG.Sens.Tt._4.AI_Output.ScaledValue;
	PG01_Local.PGSens.Tt04.Valid := PG.Sens.Tt._4.AI_Output.Status;
	PG01_Local.PGSens.Tt04.Alarm := PG.Sens.Tt._4.AI_Output.FaultLatched;
	PG01_Local.PGSens.Tt05.Value := PG.Sens.Tt._5.AI_Output.ScaledValue;
	PG01_Local.PGSens.Tt05.Valid := PG.Sens.Tt._5.AI_Output.Status;
	PG01_Local.PGSens.Tt05.Alarm := PG.Sens.Tt._5.AI_Output.FaultLatched;
	PG01_Local.PGSens.Tt06.Value := PG.Sens.Tt._6.AI_Output.ScaledValue;
	PG01_Local.PGSens.Tt06.Valid := PG.Sens.Tt._6.AI_Output.Status;
	PG01_Local.PGSens.Tt06.Alarm := PG.Sens.Tt._6.AI_Output.FaultLatched;
	PG01_Local.PGSens.Tt07.Value := PG.Sens.Tt._7.AI_Output.ScaledValue;
	PG01_Local.PGSens.Tt07.Valid := PG.Sens.Tt._7.AI_Output.Status;
	PG01_Local.PGSens.Tt07.Alarm := PG.Sens.Tt._7.AI_Output.FaultLatched;
	PG01_Local.PGSens.Tt08.Value := PG.Sens.Tt._8.AI_Output.ScaledValue;
	PG01_Local.PGSens.Tt08.Valid := PG.Sens.Tt._8.AI_Output.Status;
	PG01_Local.PGSens.Tt08.Alarm := PG.Sens.Tt._8.AI_Output.FaultLatched;
	PG01_Local.PGSens.Tt09.Value := PG.Sens.Tt._9.AI_Output.ScaledValue;
	PG01_Local.PGSens.Tt09.Valid := PG.Sens.Tt._9.AI_Output.Status;
	PG01_Local.PGSens.Tt09.Alarm := PG.Sens.Tt._9.AI_Output.FaultLatched;
	PG01_Local.PGSens.Tt10.Value := PG.Sens.Tt._10.AI_Output.ScaledValue;
	PG01_Local.PGSens.Tt10.Valid := PG.Sens.Tt._10.AI_Output.Status;
	PG01_Local.PGSens.Tt10.Alarm := PG.Sens.Tt._10.AI_Output.FaultLatched;
	PG01_Local.PGSens.Tt11.Value := PG.Sens.Tt._11.AI_Output.ScaledValue;
	PG01_Local.PGSens.Tt11.Valid := PG.Sens.Tt._11.AI_Output.Status;
	PG01_Local.PGSens.Tt11.Alarm := PG.Sens.Tt._11.AI_Output.FaultLatched;
	(* 2.10) MP01: vrednost, validnost i fault merenja nivoa/pritiska. *)
	PG01_Local.PGSens.MP01.Value := PG.Sens.MP._1.AI_Output.ScaledValue;
	PG01_Local.PGSens.MP01.Valid := PG.Sens.MP._1.AI_Output.Status;
	PG01_Local.PGSens.MP01.Alarm := PG.Sens.MP._1.AI_Output.FaultLatched;

	(* 2.11) Digitalni nivo prekidaci i prestrujni ventili: vrednost i alarm. *)
	PG01_Local.PGSens.LS01.Value := PG.Sens.LS._1.DI_Output.Value;
	PG01_Local.PGSens.LS01.Alarm := PG.Sens.LS._1.DI_Output.Alarm;
	PG01_Local.PGSens.LS02.Value := PG.Sens.LS._2.DI_Output.Value;
	PG01_Local.PGSens.LS02.Alarm := PG.Sens.LS._2.DI_Output.Alarm;
	PG01_Local.PGSens.LS03.Value := PG.Sens.LS._3.DI_Output.Value;
	PG01_Local.PGSens.LS03.Alarm := PG.Sens.LS._3.DI_Output.Alarm;
	PG01_Local.PGSens.LS04.Value := PG.Sens.LS._4.DI_Output.Value;
	PG01_Local.PGSens.LS04.Alarm := PG.Sens.LS._4.DI_Output.Alarm;
	PG01_Local.PGSens.LS05.Value := PG.Sens.LS._5.DI_Output.Value;
	PG01_Local.PGSens.LS05.Alarm := PG.Sens.LS._5.DI_Output.Alarm;
	PG01_Local.PGSens.OWF01.Value := PG.Sens.OWF._1.DI_Output.Value;
	PG01_Local.PGSens.OWF01.Alarm := PG.Sens.OWF._1.DI_Output.Alarm;
	PG01_Local.PGSens.OWF02.Value := PG.Sens.OWF._2.DI_Output.Value;
	PG01_Local.PGSens.OWF02.Alarm := PG.Sens.OWF._2.DI_Output.Alarm;
END_ACTION
```

### Data object Logical/IMA_comm_PG_BRB2/BRB2 (Simple)

#### BRB2.dat
```
; AsIMA master configuration: PT_KB_V01 -> BRB2_1
"[ROUTING_PATH]"
"/SECTION=INTERFACE"
"/CN=IF2.19"
"[PV_LIST_1]"
"/SECTION=PV"
"/SV=READ /SERVPV=PGRad_BRB2_Tx /CLNTPV=PGRad_BRB2_Rx"
"/SV=WRITE /SERVPV=PGRad_BRB2_Rx /CLNTPV=PGRad_BRB2_Tx"
"/SV=READ /SERVPV=PG01_Remote /CLNTPV=PG01_Remote"
"/SV=WRITE /SERVPV=PG01_Local /CLNTPV=PG01_Local"
```

### Alarm.typ - not listed in the package file held
```iecst
TYPE
	typAlarmState : STRUCT (* Standardno stanje jednog projektnog alarma. *)
		Active : BOOL; (* TRUE dok je fizicki ili programski uzrok trenutno prisutan. *)
		Latched : BOOL; (* TRUE od prve pojave alarma do dozvoljenog reseta. *)
		Acknowledged : BOOL; (* TRUE nakon operatorske potvrde memorisanog alarma. *)
		ResetAllowed : BOOL; (* TRUE kada aktivni uzrok vise nije prisutan. *)
		Blocking : BOOL; (* TRUE kada alarm blokira novi start ili zahteva kontrolisani stop. *)
		Code : UINT; (* Stabilan projektni alarmni kod. *)
		SourceCode : USINT; (* Lokalni FaultCode izvornog FB-a, kada postoji. *)
		Severity : USINT; (* Prioritet: 1=INFO, 2=WARNING, 3=ALARM, 4=TRIP. *)
	END_STRUCT;

	typAlarmCommand : STRUCT (* Jednociklusne komande projektnog alarmnog sistema. *)
		AcknowledgeAll : BOOL; (* Potvrda svih trenutno memorisanih alarma bez reseta opreme. *)
		ResetAlarmRecords : BOOL; (* Brisanje dozvoljenih alarmnih zapisa bez reseta opreme. *)
		ResetDevices : BOOL; (* Jednociklusni reset uredjajskih FB-ova; ne pokrece proces. *)
		ResetProcess : BOOL; (* Reset procesnog fault-a iz definisanog bezbednog stanja. *)
	END_STRUCT;

	typAlarmResetPulse : STRUCT (* Interni impulsi dostupni vlasnicima tokom celog PLC ciklusa. *)
		Devices : BOOL; (* Reset uredjaja koji ne menja procesno stanje. *)
		Process : BOOL; (* Reset procesnog fault-a koji ne pokrece sekvencu. *)
	END_STRUCT;

	typAlarmSummary : STRUCT (* Zbirni status projektnog alarmnog sistema. *)
		AnyActive : BOOL; (* Najmanje jedan alarmni uzrok je trenutno aktivan. *)
		AnyLatched : BOOL; (* Najmanje jedan alarm je memorisan. *)
		AnyUnacknowledged : BOOL; (* Najmanje jedan memorisan alarm nije potvrden. *)
		AnyTrip : BOOL; (* Najmanje jedan aktivan ili memorisan TRIP alarm postoji. *)
		RestartBlocked : BOOL; (* Novi procesni start nije dozvoljen. *)
		HighestSeverity : USINT; (* Najvisi prioritet aktivnog ili memorisanog alarma. *)
		FirstOutCode : UINT; (* Kod prvog memorisanog alarma do potpunog reseta. *)
		ActiveCount : UINT; (* Broj trenutno aktivnih alarmnih uzroka. *)
		LatchedCount : UINT; (* Broj memorisanih alarma. *)
	END_STRUCT;

	typIOModuleAlarm : STRUCT (* Status jednog fizickog IO modula. *)
		ModuleOk : BOOL; (* TRUE kada je modul prisutan i operativan. *)
		Fault : BOOL; (* TRUE kada je ModuleOk FALSE. *)
		Latched : BOOL; (* Memorisan ispad modula. *)
		Acknowledged : BOOL; (* Operatorska potvrda alarma modula. *)
		ResetAllowed : BOOL; (* TRUE kada je modul ponovo OK. *)
		Blocking : BOOL; (* TRUE kada ispad zahteva kontrolisani STOP. *)
		Code : UINT; (* Stabilan kod IO alarma. *)
	END_STRUCT;

	typPTAlarmIO : STRUCT (* Svi IO moduli Podstanice u jednoj alarmnoj grupi. *)
		X20AI4622 : typIOModuleAlarm;
		X20AI4622a : typIOModuleAlarm;
		X20AI4622b : typIOModuleAlarm;
		X20AI4622c : typIOModuleAlarm;
		X20AI4622d : typIOModuleAlarm;
		X20AO4622 : typIOModuleAlarm;
		X20AO4622a : typIOModuleAlarm;
		X20AO4622b : typIOModuleAlarm;
		X20DI9371 : typIOModuleAlarm;
		X20DI9371a : typIOModuleAlarm;
		X20DI9371b : typIOModuleAlarm;
		X20DO9322 : typIOModuleAlarm;
		X20DO9322a : typIOModuleAlarm;
		X20BC0083 : typIOModuleAlarm;
		X20PS9400 : typIOModuleAlarm;
		X20BT9100a : typIOModuleAlarm;
		X67AI1323 : typIOModuleAlarm;
		X67AI1333b : typIOModuleAlarm;
		X67DI1371_L12 : typIOModuleAlarm;
		X67DM1321_L12 : typIOModuleAlarm;
		AnyFault : BOOL;
		AnyLatched : BOOL;
		StopRequest : BOOL;
		FirstOutCode : UINT;
		FaultCount : UINT;
	END_STRUCT;

	typPTAlarmComm : STRUCT (* Alarmi komunikacije Podstanice sa udaljenim PLC-ovima. *)
		BRB2 : typAlarmState; (* Gubitak validne komunikacije sa BRB2. *)
		IEBKB1 : typAlarmState; (* Gubitak komunikacije ili heartbeat-a sa IEBKB1. *)
		BRB2RemoteFault : typAlarmState; (* Udaljeni BRB2 prijavljuje aktivan fault. *)
	END_STRUCT;

	typPTAlarmDrive : STRUCT (* Alarmi izlaznih pumpi Podstanice. *)
		PG_Pu01_VFD : typAlarmState; (* Fault frekventnog regulatora pumpe PG_Pu01. *)
		PG_Pu01_CAN : typAlarmState; (* Fault CAN komunikacije pumpe PG_Pu01. *)
		PG_Pu02_VFD : typAlarmState; (* Fault frekventnog regulatora pumpe PG_Pu02. *)
		PG_Pu02_CAN : typAlarmState; (* Fault CAN komunikacije pumpe PG_Pu02. *)
	END_STRUCT;

	typPTAlarmProcess : STRUCT (* Postojeci procesni fault kodovi Podstanice. *)
		ValveRequestConflict : typAlarmState; (* Kod 10: PG_V01 i PG_V02 istovremeno zahtevani. *)
		V01CloseTimeout : typAlarmState; (* Kod 11: PG_V01 nije zatvoren u roku. *)
		V02OpenTimeout : typAlarmState; (* Kod 12: PG_V02 nije otvoren u roku. *)
		V02CloseTimeout : typAlarmState; (* Kod 13: PG_V02 nije zatvoren u roku. *)
		V01OpenTimeout : typAlarmState; (* Kod 14: PG_V01 nije otvoren u roku. *)
		V01CloseIEBStopTimeout : typAlarmState; (* Kod 15: PG_V01 nije zatvoren pri stopu IEBKB1. *)
		IEBFlowStopTimeout : typAlarmState; (* Kod 16: IEBKB1 protok nije zaustavljen u roku. *)
		V05CloseTimeout : typAlarmState; (* Kod 17: PG_V05 nije zatvoren u roku. *)
		IEBFlowStartTimeout : typAlarmState; (* Kod 18: IEBKB1 dotok nije poceo u roku. *)
		BRB2FlowNotConfirmed : typAlarmState; (* Kod 21: BRB2 pripremni protok nije potvrden. *)
		BRB2TemperatureNotReached : typAlarmState; (* Kod 22: BRB2 pripremna temperatura nije dostignuta. *)
		PT06HighPressure : typAlarmState; (* Kod 23: PT06 pritisak je previsok tokom pripreme. *)
		TransferIEBFlowNotZero : typAlarmState; (* Kod 31: IEBKB1 protok nije pao na nulu pri transferu. *)
		TransferV05CloseTimeout : typAlarmState; (* Kod 32: PG_V05 nije zatvoren pri transferu. *)
		TransferV01CloseTimeout : typAlarmState; (* Kod 33: PG_V01 nije zatvoren pri transferu. *)
		TransferV02OpenTimeout : typAlarmState; (* Kod 34: PG_V02 nije otvoren pri transferu. *)
		TransferBRB2FlowNotConfirmed : typAlarmState; (* Kod 35: BRB2 protok nije potvrden pri transferu. *)
	END_STRUCT;

	typPTAlarmAirRelease : STRUCT (* Alarmi funkcije odzracivanja Podstanice. *)
		PG_PV03 : typAlarmState; (* Alarm odzracivanja na ulazu u Podstanicu. *)
		PG_PV04 : typAlarmState; (* Alarm odzracivanja na ulazu u prihvatni tank. *)
	END_STRUCT;

	typPTAlarm : STRUCT (* Korenski alarmni objekat PT_KB_V01 projekta. *)
		Cmd : typAlarmCommand; (* Operatorske alarmne komande. *)
		ResetPulse : typAlarmResetPulse; (* Interni reset impulsi za vlasnicke programe. *)
		Summary : typAlarmSummary; (* Zbirni status za proces i HMI. *)
		Comm : typPTAlarmComm; (* Komunikacioni alarmi. *)
		Drive : typPTAlarmDrive; (* Alarmi pogona. *)
		Process : typPTAlarmProcess; (* Procesni i sekvencni alarmi. *)
		AirRelease : typPTAlarmAirRelease; (* Alarmi odzracivanja. *)
		IO : typPTAlarmIO; (* Alarmna grupa svih fizickih IO modula. *)
	END_STRUCT;
END_TYPE
```

### PG_IO.typ - not listed in the package file held
```iecst
TYPE
	PG_type : 	STRUCT  (* Korenski tip objekta: Podstanica grejanja 1, Kursumlijska Banja *)
		Act : PG_Act_type; (* Aktuatori podstanice: pumpe, ventili *)
		Sens : PG_Sens_type; (* Senzori podstanice: pritisak, temperatura, protok, nivo *)
	END_STRUCT;
	PG_Act_type : 	STRUCT  (* Svi aktuatori podstanice PG *)
		Pu : PG_Act_Pu_type; (* Pumpe za snabdevanje potrosaca, Grundfoss CR45, METOD_DIO, 0-50 Hz *)
		PV : PG_Act_PV_type; (* Proporcionalni membranski ventili Burkert, AI/AO 4-20mA *)
		AV : PG_Act_AV_type; (* Automatski leptir ventili End Armaturen DN125 *)
		RV : PG_Act_RV_type; (* Rucni leptir ventili sa 2 krajnja prekidaca, monitoring pozicije *)
	END_STRUCT;
	PG_Sens_type : 	STRUCT  (* Svi senzori podstanice PG *)
		Pt : PG_Sens_Pt_type; (* Senzori pritiska termalne vode, Cerabar PMP23, 4-20mA *)
		Tt : PG_Sens_Tt_type; (* Senzori temperature termalne vode, Easytemp TMR35, 4-20mA *)
		MP : PG_Sens_MP_type; (* Meraci protoka termalne vode, Promag H10, 4-20mA *)
		LS : PG_Sens_LS_type; (* Nivo prekidaci u prihvatnom tanku i odzracnim cilindrima *)
		OWF : PG_Sens_OWF_type; (* Zastitni prestrujni ventili od hidraulickog udara *)
	END_STRUCT;
	PG_Act_Pu_type : 	STRUCT  (* Pumpe za snabdevanje potrosaca + vfdMain FB instance *)
		_1 : Fr_CAN_cntrl_type; (* Pumpa za snabdevanje potrosaca 01, Grundfoss CR45 *)
		_2 : Fr_CAN_cntrl_type; (* Pumpa za snabdevanje potrosaca 02, Grundfoss CR45 *)
	END_STRUCT;
	PG_Act_PV_type : 	STRUCT  (* Proporcionalni membranski ventili Burkert, AI povratni + AO komanda, 4-20mA *)
		_1 : FB_PvAiAo_Fast; (* Ulazni regulacioni ventil 1 - prihvatni tank, DN050 NC *)
		_2 : FB_PvAiAo_Fast; (* Ulazni regulacioni ventil 2 - prihvatni tank, DN050 NC *)
		_3 : FB_PvAiAo_Fast; (* Odzracni ventil na ulazu termalne vode u kotlarnicu, DN025 NC *)
		_4 : FB_PvAiAo_Fast; (* Odzracni ventil na ulazu termalne vode u prihvatni tank, DN025 NC *)
		_5 : FB_PvAiAo_Fast; (* PG_PV05 - regulacija pritiska PT06 i drenazno preispiranje BRB2 grane. *)
	END_STRUCT;
	PG_Act_AV_type : 	STRUCT  (* Automatski leptir ventili End Armaturen DN125, bistabilni i spring-return *)
		_1 : FB_V_EMV; (* Elektromotorni bistabilni, CmdOpen + CmdClose, OpenMaxTime=20s *)
		_2 : FB_V_EMV; (* Elektromotorni bistabilni, CmdOpen + CmdClose, OpenMaxTime=20s *)
		_3 : FB_V_ON_OFF_FB; (* Pneumatski NC spring-return, samo CmdOpen, OpenMaxTime=10s *)
		_4 : FB_V_ON_OFF_FB; (* Pneumatski NC spring-return, samo CmdOpen, OpenMaxTime=10s *)
		_5 : FB_V_ON_OFF_FB; (* Pneumatski NC spring-return, samo CmdOpen, OpenMaxTime=10s *)
		_6 : FB_V_ON_OFF_FB; (* Pneumatski NC spring-return, samo CmdOpen, OpenMaxTime=10s *)
		_7 : FB_V_ON_OFF_FB; (* Pneumatski NC spring-return, samo CmdOpen, OpenMaxTime=10s *)
	END_STRUCT;
	PG_Act_RV_type : 	STRUCT  (* Rucni leptir ventili NIOB FLUID / End Armaturen, monitoring 2 krajnja prekidaca *)
		_19 : FB_HV_2LS; (* Rucni ventil posle membranskog ventila PG_PV01 *)
		_21 : FB_HV_2LS; (* Rucni ventil posle membranskog ventila PG_PV02 *)
		_22 : FB_HV_2LS; (* Drenazni total ventil na dnu prihvatnog tanka *)
		_23 : FB_HV_2LS; (* Ulaz u Pumpu PG_Pu01 *)
		_24 : FB_HV_2LS; (* Ulaz u Pumpu PG_Pu02 *)
		_25 : FB_HV_2LS; (* Bajpasni izlaz iz tanka ka instalaciji za izbacivanje gasa van kotlarnice *)
		_26 : FB_HV_2LS; (* Ulaz u vakuum pumpu *)
		_27 : FB_HV_2LS; (* Izlaz iz vakuum pumpe ka instalaciji za izbacivanje gasa van kotlarnice *)
	END_STRUCT;
	PG_Sens_Pt_type : 	STRUCT  (* Senzori pritiska termalne vode, 9x FBAI01_DI01, Cerabar PMP23, 4-20mA, opseg -1..9 bar / -100..300 mbar / -1..14 bar *)
		_0_0 : FBAI01_DI01; (* Pritisak komprimovanog vazduha, opseg -1..14 bar *)
		_1 : FBAI01_DI01; (* Pritisak termalne vode na ulazu u podstanicu *)
		_2 : FBAI01_DI01; (* Pritisak termalne vode posle streinera grubih filtera *)
		_3 : FBAI01_DI01; (* Pritisak termalne vode posle velikog izmenjivaca *)
		_4 : FBAI01_DI01; (* Pritisak termalne vode na ulazu u prihvatni tank *)
		_5 : FBAI01_DI01; (* Pritisak na potisu transportnih pumpi *)
		_6 : FBAI01_DI01; (* PT_PG_06 - pritisak dolazne BRB2 magistrale pre PG_V02, opseg -1..9 bar. *)
		_NS1 : FBAI01_DI01; (* Pritisak na dnu prihvatnog tanka [mbar] *)
		_NS2 : FBAI01_DI01; (* Pritisak na vrhu prihvatnog tanka [mbar] *)
	END_STRUCT;
	PG_Sens_Tt_type : 	STRUCT  (* Senzori temperature termalne vode, Easytemp TMR35, 4-20mA, opseg 0-120 degC *)
		_1 : FBAI01_DI01; (* TT_PG_01 - ulaz u veliki razmenjivac PGRT01. *)
		_2 : FBAI01_DI01; (* TT_PG_02 - temperatura na ulazu u prihvatni tank. *)
		_3 : FBAI01_DI01; (* TT_PG_03 - temperatura u prihvatnom tanku. *)
		_4 : FBAI01_DI01; (* TT_PG_04 - izlaz iz velikog razmenjivaca PGRT01. *)
		_5 : FBAI01_DI01; (* TT_PG_05 - ulaz u mali razmenjivac PGRT02. *)
		_6 : FBAI01_DI01; (* TT_PG_06 - izlaz iz malog razmenjivaca PGRT02. *)
		_7 : FBAI01_DI01; (* TT_PG_07 - drenazni vod za potvrdu zavrsetka preispiranja. *)
		_8 : FBAI01_DI01; (* TT_PG_08 - Ulaz tehnicke vode u direktni iztmenbjivac toplote*)
		_9 : FBAI01_DI01; (* TT_PG_09 - Izlaz tehnicke vode iz direktnog iztmenbjivaca toplote*)
		_10 : FBAI01_DI01; (* TT_PG_10 - Ulaz tsanitarne vode u direktni iztmenbjivac toplote*)
		_11 : FBAI01_DI01; (* TT_PG_11 - Izlaz sanitarne vode iz direktnog iztmenbjivaca toplote*)
	END_STRUCT;
	PG_Sens_MP_type : 	STRUCT  (* Meraci protoka, 1x FBAI01_DI01, Promag H10 DN065, 4-20mA, opseg 0-72 m3/h *)
		_1 : FBAI01_DI01; (* MeraÄ protoka na potisu tople termalne vode ka potrosacima *)
	END_STRUCT;
	PG_Sens_LS_type : 	STRUCT  (* Nivo prekidaci Liquipoint FTW23, 5x FB_DI, detekcija tecnosti u prihvatnom tanku i odzracnim cilindrima *)
		_1 : FB_DI; (* Nizak nivo vode u prihvatnom tanku za rad pumpi *)
		_2 : FB_DI; (* Donji nivo u odzracnom cilindru na ulazu vode u podstanicu *)
		_3 : FB_DI; (* Gornji nivo u odzracnom cilindru na ulazu vode u podstanicu *)
		_4 : FB_DI; (* Donji nivo u odzracnom cilindru na ulazu vode u prihvatni tank *)
		_5 : FB_DI; (* Gornji nivo u odzracnom cilindru na ulazu vode u prihvatni tank *)
	END_STRUCT;
	PG_Sens_OWF_type : 	STRUCT  (* Zastitni prestrujni ventili NIOB FLUID 5371 DN050, 2x FB_DI, zastita od hidraulickog udara *)
		_1 : FB_DI; (* Zastitni prestrujni ventil od hidraulickog udara 1 *)
		_2 : FB_DI; (* Zastitni prestrujni ventil od hidraulickog udara 2 *)
	END_STRUCT;
	Fr_CAN_cntrl_type : 	STRUCT  (* Komande, granice i CAN telemetrija glavne pumpe RB2_01. *)
		Enable : BOOL; (* Dozvola CAN pogona; vodi ATV stanje iz Standby ka Ready. *)
		Start : BOOL; (* Komanda rada CAN pogona; vodi ATV stanje iz Ready ka InRun. *)
		Alarm_FR : BOOL; (* TRUE = aktivan fault frekventnog regulatora. *)
		Alarm_CAN : BOOL; (* TRUE = aktivan alarm CAN komunikacije sa pogonom. *)
		Reset_Alarm : BOOL; (* Jednociklusni zahtev za reset fault-a pogona. *)
		Node_status : UINT; (* Sirovi CANopen status komunikacionog cvora RB2_01. *)
		FR_min : REAL; (* Deklarisana donja granica frekventnog zahteva [Hz]. *)
		FR_max : REAL; (* Deklarisana gornja granica frekventnog zahteva [Hz]. *)
		Motor_Snaga : REAL; (*Snaga motora u kW *)
		Motor_Nominalna_Snaga : REAL; (*Nominalna snaga motora u kW *)
		Motor_Struja : REAL; (*Struja motora u A *)
		FR_set : REAL; (*Zadata frekvenca u Hz*)
		Ostvarena_brzina : REAL; (*Ostvarena brzina motora - control effort u Hz*)
		Status_inRun : BOOL; (*Status da je fr u In run modu*)
		CAN_FB : FbCanAtv; (* Vlasnicka instanca CANopen upravljanja ATV pogonom RB2_01. *)
		U_int : U_struct_int; (* Sirove CAN vrednosti linijskih napona u desetinkama volta. *)
		U_real : U_struct_real; (* Preracunati linijski naponi za HMI i dijagnostiku [V]. *)
	END_STRUCT;
	U_struct_real : 	STRUCT  (* Preracunati trofazni linijski naponi pogona [V]. *)
		U_srednje : REAL; (* Srednja vrednost linijskih napona [V]. *)
		U_12 : REAL; (* Linijski napon faza L1-L2 [V]. *)
		U_23 : REAL; (* Linijski napon faza L2-L3 [V]. *)
		U_31 : REAL; (* Linijski napon faza L3-L1 [V]. *)
	END_STRUCT;
	U_struct_int : 	STRUCT  (* Sirovi CAN registri trofaznih linijskih napona [0.1 V]. *)
		U_srednje : UINT; (* Sirova srednja vrednost linijskih napona [0.1 V]. *)
		U_12 : INT; (* Sirovi linijski napon faza L1-L2 [0.1 V]. *)
		U_23 : INT; (* Sirovi linijski napon faza L2-L3 [0.1 V]. *)
		U_31 : INT; (* Sirovi linijski napon faza L3-L1 [0.1 V]. *)
	END_STRUCT;
END_TYPE
```

### PGRad_Communication.typ - not listed in the package file held
```iecst
TYPE
	typVezaPGRadBRB2 : 	STRUCT  (* Dvosmerni procesni ugovor: PT pise komande, BRB2 pise statuse. *)
			RadKaPodstanici : BOOL; (* PT izbor rute BRB2 ka podstanici; prihvata se samo u BRB2 standby. *)
			ManualMode : BOOL; (* Dozvola servisnog rucnog rezima. *)
			ManualSequence : USINT; (* Izabrana servisna sekvenca. *)
			ManualStart : BOOL; (* Impuls za pokretanje servisne sekvence. *)
			ManualStop : BOOL; (* Impuls za bezbedan prekid servisne sekvence. *)
			ManualNextStep : BOOL; (* Impuls za sledeci dozvoljeni podkorak. *)
			ManualAbort : BOOL; (* Impuls za povratak u Standby. *)
			CommandCounter : UDINT; (* Monotoni PT brojac za BRB2 watchdog komandi. *)
			ZahtevStarta : BOOL; (* PT zahtev BRB2 za pripremu i start bunarske pumpe. *)
			ZahtevZaustavljanja : BOOL; (* PT zahtev BRB2 za kontrolisano zaustavljanje. *)
			VentiliPodstaniceZatvoreni : BOOL; (* PT potvrda zatvorenosti PG_PV01, PG_PV02 i PG_PV05. *)
			PritisakIEBKB1 : REAL; (* PT prosledjuje stvarni pritisak IEBKB1 odredista [bar]. *)
			PodstanicaURezimuRada : BOOL; (* PT tank je na nivou i izabrana izlazna pumpa je stvarno u radu. *)
			RegulationMode : USINT; (* PT izbor BRB2 petlje preko AsIMA: 0=neaktivna, 1=protok, 2=nivo, 3=temperatura. *)
			RegulationPV : REAL; (* PT prosledjuje procesnu vrednost aktivne petlje. *)
			RegulationSP : REAL; (* PT prosledjuje zadatu vrednost aktivne petlje. *)
			RegulationPVValid : BOOL; (* PT potvrda validnosti aktivne procesne vrednosti. *)
			RegulationInvert : BOOL; (* PT zahtev za obrtanje smera regulacije. *)
			NivoPrihvatniSud : REAL; (* Nivo prihvatnog suda koji se salje BRB2 kao PV moda 2 [m]. *)
			StatusCounter : UDINT; (* Monotoni BRB2 brojac za PT watchdog statusa. *)
			BRB2Fault : BOOL; (* Zbirni fault aktivne BRB2 pumpe ili regulatora. *)
			BRB2FaultCode : USINT; (* Stabilan kod BRB2 fault uzroka za Podstanicu. *)
			RegulationPVFault : BOOL; (* Aktivni PV nije validan duze od dozvoljenog vremena. *)
			PumpaAktivna : BOOL; (* BRB2 stvarna potvrda da je RB2_01 u InRun stanju. *)
			IspiranjeProtokDostignut : BOOL; (* BRB2 stvarni protok je dostigao ProtokIspiranja. *)
			IspiranjeMinTrajanjeDostignuto : BOOL; (* BRB2 je na ProtokIspiranja najmanje T_IspiranjeMin. *)
			StopSPDostignut : BOOL; (* BRB2 potvrda dostignutog FR_MinZeroFlow. *)
			RB2V01Zatvoren : BOOL; (* BRB2 potvrda zatvorenog RB2_V01 za IEBKB1 granu. *)
			RB2V02Zatvoren : BOOL; (* BRB2 potvrda zatvorenog RB2_V02. *)
		END_STRUCT;
		typBRB2CommWatchdog : 	STRUCT (* Lokalna memorija i validnost watchdog-a udaljenog brojaca. *)
			LastCounter : UDINT; (* Poslednji primljeni udaljeni brojac. *)
			ReceivedOnce : BOOL; (* TRUE nakon prve registrovane promene udaljenog brojaca. *)
			ReceiveTimeout : TON; (* Timeout bez promene udaljenog brojaca. *)
			Valid : BOOL; (* TRUE dok se udaljeni brojac menja unutar 5 s. *)
		END_STRUCT;
		typIEBKB1PreparedInterface : 	STRUCT  (* Lokalno pripremljen ugovor; jos nije deo postojeceg IEB wire-layout-a. *)
			Enable : BOOL; (* Dozvola koriscenja prosirenog IEBKB1 ugovora. *)
			InterfaceReady : BOOL; (* Verzija udaljenog PLC-a podrzava sva sledeca polja. *)
			CommValid : BOOL; (* AsIMA komunikacija je validna. *)
			HeartbeatValid : BOOL; (* Heartbeat se menja unutar dozvoljenog vremena. *)
			HeartbeatCounter : UDINT; (* Poslednji primljeni heartbeat brojac. *)
			Fault : BOOL; (* IEBKB1 prijavljuje aktivnu gresku. *)
			CommandAccepted : BOOL; (* IEBKB1 je prihvatio poslednju procesnu komandu. *)
			PumpRunning : BOOL; (* IEBKB1 potvrda stvarnog rada pumpe. *)
			FlowValid : BOOL; (* IEBKB1 potvrda validnog merenja protoka. *)
		END_STRUCT;
END_TYPE
```

### PGRad_HMI.typ - not listed in the package file held
```iecst
TYPE
	typPGRadTrendCursor : 	STRUCT (* HMI stanje vremenske ose, kursora i procesnih vrednosti trenda Podstanice. *)
			Position : REAL; (* Normalizovana pozicija kursora: 0.0 = levo, 1.0 = desno. *)
			Time : UDINT; (* Proteklo vreme od pocetka trend zapisa na poziciji kursora [ms]. *)
			RecordingStart : DATE_AND_TIME; (* Apsolutno vreme pocetka referentnog trend zapisa. *)
			DateTime : DATE_AND_TIME; (* Apsolutni datum i vreme uzorka na poziciji kursora. *)
			ViewStart : DATE_AND_TIME; (* Leva granica trenutno prikazanog vremenskog prozora. *)
			ViewSpan : DINT; (* Sirina prikazanog vremenskog prozora [s]. *)
			AxisMode : UINT; (* VC time-scale mod: 0 = zadati prozor bez automatskog pomeranja. *)
			PreviousViewSpan : DINT; (* Prethodna sirina prozora za promenu zoom-a bez skoka. *)
			FollowNow : BOOL; (* TRUE = desna ivica prozora prati trenutno vreme. *)
			CmdBack : BOOL; (* Jednokratni zahtev za prethodni vremenski prozor. *)
			CmdForward : BOOL; (* Jednokratni zahtev za sledeci vremenski prozor. *)
			CmdNow : BOOL; (* Jednokratni zahtev za povratak na najnovije podatke. *)
			AxisTime0 : DATE_AND_TIME; (* Pocetak prikazanog vremenskog prozora. *)
			AxisTime1 : DATE_AND_TIME; (* Prva unutrasnja vremenska oznaka ose. *)
			AxisTime2 : DATE_AND_TIME; (* Druga unutrasnja vremenska oznaka ose. *)
			AxisTime3 : DATE_AND_TIME; (* Treca unutrasnja vremenska oznaka ose. *)
			AxisTime4 : DATE_AND_TIME; (* Cetvrta unutrasnja vremenska oznaka ose. *)
			AxisTime5 : DATE_AND_TIME; (* Peta unutrasnja vremenska oznaka ose. *)
			AxisTime6 : DATE_AND_TIME; (* Sesta unutrasnja vremenska oznaka ose. *)
			AxisTime7 : DATE_AND_TIME; (* Sedma unutrasnja vremenska oznaka ose. *)
			AxisTime8 : DATE_AND_TIME; (* Kraj prikazanog vremenskog prozora. *)
			Status : UINT; (* VC status trend kursora; bit 10 oznacava validan Cursor 1. *)
			Nivo : REAL; (* Nivo prihvatnog tanka na poziciji kursora [m]. *)
			Pritisak : REAL; (* PT05 pritisak potisa pumpe na poziciji kursora [bar]. *)
			Protok : REAL; (* Protok ka bazenima na poziciji kursora [l/s]. *)
			TT01 : REAL; (* Temperatura TT01 na poziciji kursora [degC]. *)
			TT03 : REAL; (* Temperatura u prihvatnom tanku TT03 na poziciji kursora [degC]. *)
			TT04 : REAL; (* Temperatura TT04 na poziciji kursora [degC]. *)
			TT05 : REAL; (* Temperatura TT05 na poziciji kursora [degC]. *)
			TT06 : REAL; (* Temperatura TT06 na poziciji kursora [degC]. *)
		END_STRUCT;
END_TYPE
```
